LIN {X 0,Y 530.989,Z 469.465,A -85,B 0,C 180,E1 -4213.071,E2 -4213.071} C_VEL
LIN {X 0,Y 531.043,Z 469.464,A -85,B 0,C 180,E1 -4215.436,E2 -4215.436} C_VEL
LIN {X 0,Y 531.04,Z 469.456,A -85,B 0,C 180,E1 -4218.55,E2 -4218.55} C_VEL
LIN {X 0,Y 531.062,Z 469.46,A -85,B 0,C 180,E1 -4221.629,E2 -4221.629} C_VEL
LIN {X 0,Y 531.124,Z 469.446,A -85,B 0,C 180,E1 -4224.685,E2 -4224.685} C_VEL
LIN {X 0,Y 531.144,Z 469.448,A -85,B 0,C 180,E1 -4227.725,E2 -4227.725} C_VEL
LIN {X 0,Y 531.154,Z 469.442,A -85,B 0,C 180,E1 -4230.758,E2 -4230.758} C_VEL
LIN {X 0,Y 531.108,Z 469.451,A -85,B 0,C 180,E1 -4233.034,E2 -4233.034} C_VEL
LIN {X 0,Y 531.078,Z 469.452,A -85,B 0,C 180,E1 -4236.077,E2 -4236.077} C_VEL
LIN {X 0,Y 531.058,Z 469.454,A -85,B 0,C 180,E1 -4238.37,E2 -4238.37} C_VEL
LIN {X 0,Y 531.054,Z 469.459,A -85,B 0,C 180,E1 -4241.672,E2 -4241.672} C_VEL
LIN {X 0,Y 531.033,Z 469.46,A -85,B 0,C 180,E1 -4244.956,E2 -4244.956} C_VEL
LIN {X 0,Y 531.019,Z 469.463,A -85,B 0,C 180,E1 -4247.722,E2 -4247.722} C_VEL
LIN {X 0,Y 531.002,Z 469.464,A -85,B 0,C 180,E1 -4250.938,E2 -4250.938} C_VEL
LIN {X 0,Y 530.982,Z 469.463,A -85,B 0,C 180,E1 -4254.224,E2 -4254.224} C_VEL
LIN {X 0,Y 531.006,Z 469.461,A -85,B 0,C 180,E1 -4256.744,E2 -4256.744} C_VEL
LIN {X 0,Y 530.984,Z 469.472,A -85,B 0,C 180,E1 -4259.323,E2 -4259.323} C_VEL
LIN {X 0,Y 530.968,Z 469.465,A -85,B 0,C 180,E1 -4262.1,E2 -4262.1} C_VEL
LIN {X 0,Y 530.972,Z 469.467,A -85,B 0,C 180,E1 -4264.851,E2 -4264.851} C_VEL
LIN {X 0,Y 530.968,Z 469.472,A -85,B 0,C 180,E1 -4267.508,E2 -4267.508} C_VEL
LIN {X 0,Y 530.986,Z 469.463,A -85,B 0,C 180,E1 -4270.433,E2 -4270.433} C_VEL
LIN {X 0,Y 530.973,Z 469.473,A -85,B 0,C 180,E1 -4273.282,E2 -4273.282} C_VEL
LIN {X 0,Y 530.985,Z 469.467,A -85,B 0,C 180,E1 -4275.622,E2 -4275.622} C_VEL
LIN {X 0,Y 530.995,Z 469.462,A -85,B 0,C 180,E1 -4278.565,E2 -4278.565} C_VEL
LIN {X 0,Y 530.961,Z 469.471,A -85,B 0,C 180,E1 -4281.53,E2 -4281.53} C_VEL
LIN {X 0,Y 530.959,Z 469.466,A -85,B 0,C 180,E1 -4284.38,E2 -4284.38} C_VEL
LIN {X 0,Y 530.97,Z 469.472,A -85,B 0,C 180,E1 -4287.134,E2 -4287.134} C_VEL
LIN {X 0,Y 530.972,Z 469.467,A -85,B 0,C 180,E1 -4289.803,E2 -4289.803} C_VEL
LIN {X 0,Y 531.015,Z 469.461,A -85,B 0,C 180,E1 -4292.468,E2 -4292.468} C_VEL
LIN {X 0,Y 531.043,Z 469.626,A -85,B 0,C 180,E1 -4294.433,E2 -4294.433} C_VEL
LIN {X 0,Y 532.717,Z 478.043,A -85,B 0,C 180,E1 -4295.699,E2 -4295.699} C_VEL
LIN {X 0,Y 532.591,Z 490.919,A -85,B 0,C 180,E1 -4297.5,E2 -4297.5} C_VEL
LIN {X 0,Y 532.133,Z 510.715,A -85,B 0,C 180,E1 -4300.319,E2 -4300.319} C_VEL
LIN {X 0,Y 531.751,Z 532.106,A -85,B 0,C 180,E1 -4303.294,E2 -4303.294} C_VEL
LIN {X 0,Y 531.511,Z 544.809,A -85,B 0,C 180,E1 -4305.09,E2 -4305.09} C_VEL
LIN {X 0,Y 532.811,Z 554.136,A -85,B 0,C 180,E1 -4305.262,E2 -4305.262} C_VEL
LIN {X 0,Y 532.416,Z 652.888,A -85,B 0,C 180,E1 -4306.62,E2 -4306.62} C_VEL
LIN {X 0,Y 532.247,Z 665.054,A -85,B 0,C 180,E1 -4306.907,E2 -4306.907} C_VEL
LIN {X 0,Y 532.045,Z 678.792,A -85,B 0,C 180,E1 -4307.411,E2 -4307.411} C_VEL
LIN {X 0,Y 531.781,Z 689.648,A -85,B 0,C 180,E1 -4307.956,E2 -4307.956} C_VEL
LIN {X 0,Y 531.654,Z 697.634,A -85,B 0,C 180,E1 -4308.447,E2 -4308.447} C_VEL
LIN {X 0,Y 531.413,Z 706.954,A -85,B 0,C 180,E1 -4309.137,E2 -4309.137} C_VEL
LIN {X 0,Y 531.231,Z 713.575,A -85,B 0,C 180,E1 -4309.712,E2 -4309.712} C_VEL
LIN {X 0,Y 531.071,Z 721.12,A -85,B 0,C 180,E1 -4310.478,E2 -4310.478} C_VEL
LIN {X 0,Y 530.921,Z 727.6,A -85,B 0,C 180,E1 -4311.244,E2 -4311.244} C_VEL
LIN {X 0,Y 530.76,Z 734.405,A -85,B 0,C 180,E1 -4312.2,E2 -4312.2} C_VEL
LIN {X 0,Y 530.643,Z 740.091,A -85,B 0,C 180,E1 -4313.154,E2 -4313.154} C_VEL
LIN {X 0,Y 530.609,Z 745.619,A -85,B 0,C 180,E1 -4314.299,E2 -4314.299} C_VEL
LIN {X 0,Y 530.462,Z 749.968,A -85,B 0,C 180,E1 -4315.441,E2 -4315.441} C_VEL
LIN {X 0,Y 530.516,Z 752.339,A -85,B 0,C 180,E1 -4316.202,E2 -4316.202} C_VEL
LIN {X 0,Y 530.457,Z 754.172,A -85,B 0,C 180,E1 -4316.962,E2 -4316.962} C_VEL
LIN {X 0,Y 530.361,Z 756.638,A -85,B 0,C 180,E1 -4318.481,E2 -4318.481} C_VEL
LIN {X 0,Y 530.344,Z 757.24,A -85,B 0,C 180,E1 -4319.241,E2 -4319.241} C_VEL
LIN {X 0,Y 530.344,Z 757.307,A -85,B 0,C 180,E1 -4320.759,E2 -4320.759} C_VEL
LIN {X 0,Y 530.361,Z 756.712,A -85,B 0,C 180,E1 -4321.519,E2 -4321.519} C_VEL
LIN {X 0,Y 530.457,Z 754.383,A -85,B 0,C 180,E1 -4323.038,E2 -4323.038} C_VEL
LIN {X 0,Y 530.522,Z 751.5,A -85,B 0,C 180,E1 -4324.178,E2 -4324.178} C_VEL
LIN {X 0,Y 530.523,Z 747.581,A -85,B 0,C 180,E1 -4325.321,E2 -4325.321} C_VEL
LIN {X 0,Y 530.552,Z 743.338,A -85,B 0,C 180,E1 -4326.305,E2 -4326.305} C_VEL
LIN {X 0,Y 530.678,Z 737.337,A -85,B 0,C 180,E1 -4327.419,E2 -4327.419} C_VEL
LIN {X 0,Y 530.843,Z 731.101,A -85,B 0,C 180,E1 -4328.374,E2 -4328.374} C_VEL
LIN {X 0,Y 530.978,Z 723.591,A -85,B 0,C 180,E1 -4329.331,E2 -4329.331} C_VEL
LIN {X 0,Y 531.199,Z 716.488,A -85,B 0,C 180,E1 -4330.096,E2 -4330.096} C_VEL
LIN {X 0,Y 531.382,Z 708.045,A -85,B 0,C 180,E1 -4330.863,E2 -4330.863} C_VEL
LIN {X 0,Y 531.562,Z 700.597,A -85,B 0,C 180,E1 -4331.439,E2 -4331.439} C_VEL
LIN {X 0,Y 531.786,Z 691.155,A -85,B 0,C 180,E1 -4332.047,E2 -4332.047} C_VEL
LIN {X 0,Y 531.939,Z 680.692,A -85,B 0,C 180,E1 -4332.592,E2 -4332.592} C_VEL
LIN {X 0,Y 532.174,Z 669.962,A -85,B 0,C 180,E1 -4333.022,E2 -4333.022} C_VEL
LIN {X 0,Y 532.375,Z 656.359,A -85,B 0,C 180,E1 -4333.406,E2 -4333.406} C_VEL
LIN {X 0,Y 532.522,Z 634.145,A -85,B 0,C 180,E1 -4333.742,E2 -4333.742} C_VEL
LIN {X 0,Y 532.733,Z 552.911,A -85,B 0,C 180,E1 -4334.844,E2 -4334.844} C_VEL
LIN {X 0,Y 531.512,Z 544.794,A -85,B 0,C 180,E1 -4335.007,E2 -4335.007} C_VEL
LIN {X 0,Y 531.862,Z 525.613,A -85,B 0,C 180,E1 -4337.693,E2 -4337.693} C_VEL
LIN {X 0,Y 532.252,Z 507.489,A -85,B 0,C 180,E1 -4340.244,E2 -4340.244} C_VEL
LIN {X 0,Y 532.568,Z 484.627,A -85,B 0,C 180,E1 -4343.322,E2 -4343.322} C_VEL
LIN {X 0,Y 532.427,Z 476.639,A -85,B 0,C 180,E1 -4344.384,E2 -4344.384} C_VEL
LIN {X 0,Y 531.039,Z 469.463,A -85,B 0,C 180,E1 -4345.423,E2 -4345.423} C_VEL
LIN {X 0,Y 531,Z 469.469,A -85,B 0,C 180,E1 -4348.455,E2 -4348.455} C_VEL
LIN {X 0,Y 530.96,Z 469.474,A -85,B 0,C 180,E1 -4351.079,E2 -4351.079} C_VEL
LIN {X 0,Y 530.99,Z 469.465,A -85,B 0,C 180,E1 -4353.773,E2 -4353.773} C_VEL
LIN {X 0,Y 530.958,Z 469.475,A -85,B 0,C 180,E1 -4356.558,E2 -4356.558} C_VEL
LIN {X 0,Y 530.991,Z 469.464,A -85,B 0,C 180,E1 -4359.443,E2 -4359.443} C_VEL
LIN {X 0,Y 530.98,Z 469.471,A -85,B 0,C 180,E1 -4362.457,E2 -4362.457} C_VEL
LIN {X 0,Y 530.991,Z 469.463,A -85,B 0,C 180,E1 -4365.621,E2 -4365.621} C_VEL
LIN {X 0,Y 531,Z 469.469,A -85,B 0,C 180,E1 -4368.565,E2 -4368.565} C_VEL
LIN {X 0,Y 530.96,Z 469.467,A -85,B 0,C 180,E1 -4371.529,E2 -4371.529} C_VEL
LIN {X 0,Y 530.982,Z 469.471,A -85,B 0,C 180,E1 -4374.382,E2 -4374.382} C_VEL
LIN {X 0,Y 530.975,Z 469.466,A -85,B 0,C 180,E1 -4377.134,E2 -4377.134} C_VEL
LIN {X 0,Y 530.989,Z 469.467,A -85,B 0,C 180,E1 -4379.804,E2 -4379.804} C_VEL
LIN {X 0,Y 531.017,Z 469.468,A -85,B 0,C 180,E1 -4382.467,E2 -4382.467} C_VEL
LIN {X 0,Y 531.078,Z 469.651,A -85,B 0,C 180,E1 -4384.92,E2 -4384.92} C_VEL
LIN {X 0,Y 533.286,Z 479.428,A -85,B 0,C 180,E1 -4386.3,E2 -4386.3} C_VEL
LIN {X 0,Y 532.933,Z 495.381,A -85,B 0,C 180,E1 -4388.331,E2 -4388.331} C_VEL
LIN {X 0,Y 532.3,Z 520.903,A -85,B 0,C 180,E1 -4391.526,E2 -4391.526} C_VEL
LIN {X 0,Y 532.17,Z 524.017,A -85,B 0,C 180,E1 -4391.91,E2 -4391.91} C_VEL
LIN {X 0,Y 533.88,Z 534.449,A -85,B 0,C 180,E1 -4392.114,E2 -4392.114} C_VEL
LIN {X 0,Y 533.255,Z 662.06,A -85,B 0,C 180,E1 -4393.859,E2 -4393.859} C_VEL
LIN {X 0,Y 533.024,Z 676.356,A -85,B 0,C 180,E1 -4394.202,E2 -4394.202} C_VEL
LIN {X 0,Y 532.797,Z 690.478,A -85,B 0,C 180,E1 -4394.703,E2 -4394.703} C_VEL
LIN {X 0,Y 532.549,Z 702.8,A -85,B 0,C 180,E1 -4395.283,E2 -4395.283} C_VEL
LIN {X 0,Y 532.13,Z 715.67,A -85,B 0,C 180,E1 -4396.052,E2 -4396.052} C_VEL
LIN {X 0,Y 531.813,Z 727.305,A -85,B 0,C 180,E1 -4396.92,E2 -4396.92} C_VEL
LIN {X 0,Y 531.463,Z 738.313,A -85,B 0,C 180,E1 -4397.917,E2 -4397.917} C_VEL
LIN {X 0,Y 531.235,Z 747.706,A -85,B 0,C 180,E1 -4398.94,E2 -4398.94} C_VEL
LIN {X 0,Y 530.935,Z 756.556,A -85,B 0,C 180,E1 -4400.091,E2 -4400.091} C_VEL
LIN {X 0,Y 530.775,Z 765.034,A -85,B 0,C 180,E1 -4401.433,E2 -4401.433} C_VEL
LIN {X 0,Y 530.586,Z 771.863,A -85,B 0,C 180,E1 -4402.771,E2 -4402.771} C_VEL
LIN {X 0,Y 530.584,Z 777.961,A -85,B 0,C 180,E1 -4404.299,E2 -4404.299} C_VEL
LIN {X 0,Y 530.449,Z 781.444,A -85,B 0,C 180,E1 -4405.44,E2 -4405.44} C_VEL
LIN {X 0,Y 530.452,Z 784.832,A -85,B 0,C 180,E1 -4406.962,E2 -4406.962} C_VEL
LIN {X 0,Y 530.356,Z 786.835,A -85,B 0,C 180,E1 -4408.481,E2 -4408.481} C_VEL
LIN {X 0,Y 530.341,Z 787.5,A -85,B 0,C 180,E1 -4410,E2 -4410} C_VEL
LIN {X 0,Y 530.356,Z 786.836,A -85,B 0,C 180,E1 -4411.519,E2 -4411.519} C_VEL
LIN {X 0,Y 530.452,Z 784.836,A -85,B 0,C 180,E1 -4413.038,E2 -4413.038} C_VEL
LIN {X 0,Y 530.449,Z 781.446,A -85,B 0,C 180,E1 -4414.56,E2 -4414.56} C_VEL
LIN {X 0,Y 530.56,Z 776.567,A -85,B 0,C 180,E1 -4416.083,E2 -4416.083} C_VEL
LIN {X 0,Y 530.641,Z 770.053,A -85,B 0,C 180,E1 -4417.611,E2 -4417.611} C_VEL
LIN {X 0,Y 530.818,Z 762.803,A -85,B 0,C 180,E1 -4418.95,E2 -4418.95} C_VEL
LIN {X 0,Y 531.018,Z 753.821,A -85,B 0,C 180,E1 -4420.293,E2 -4420.293} C_VEL
LIN {X 0,Y 531.311,Z 744.391,A -85,B 0,C 180,E1 -4421.444,E2 -4421.444} C_VEL
LIN {X 0,Y 531.585,Z 733.95,A -85,B 0,C 180,E1 -4422.503,E2 -4422.503} C_VEL
LIN {X 0,Y 531.956,Z 722.424,A -85,B 0,C 180,E1 -4423.465,E2 -4423.465} C_VEL
LIN {X 0,Y 532.29,Z 709.619,A -85,B 0,C 180,E1 -4424.333,E2 -4424.333} C_VEL
LIN {X 0,Y 532.625,Z 696.975,A -85,B 0,C 180,E1 -4425.008,E2 -4425.008} C_VEL
LIN {X 0,Y 532.891,Z 683.069,A -85,B 0,C 180,E1 -4425.579,E2 -4425.579} C_VEL
LIN {X 0,Y 533.151,Z 668.504,A -85,B 0,C 180,E1 -4426.002,E2 -4426.002} C_VEL
LIN {X 0,Y 533.291,Z 653.936,A -85,B 0,C 180,E1 -4426.263,E2 -4426.263} C_VEL
LIN {X 0,Y 533.831,Z 534.167,A -85,B 0,C 180,E1 -4427.883,E2 -4427.883} C_VEL
LIN {X 0,Y 532.175,Z 524.02,A -85,B 0,C 180,E1 -4428.083,E2 -4428.083} C_VEL
LIN {X 0,Y 532.831,Z 498.464,A -85,B 0,C 180,E1 -4431.268,E2 -4431.268} C_VEL
LIN {X 0,Y 533.425,Z 481.072,A -85,B 0,C 180,E1 -4433.488,E2 -4433.488} C_VEL
LIN {X 0,Y 532.289,Z 474.884,A -85,B 0,C 180,E1 -4434.352,E2 -4434.352} C_VEL
LIN {X 0,Y 531.038,Z 469.465,A -85,B 0,C 180,E1 -4435.161,E2 -4435.161} C_VEL
LIN {X 0,Y 531.018,Z 469.468,A -85,B 0,C 180,E1 -4437.596,E2 -4437.596} C_VEL
LIN {X 0,Y 530.978,Z 469.468,A -85,B 0,C 180,E1 -4440.645,E2 -4440.645} C_VEL
LIN {X 0,Y 530.989,Z 469.47,A -85,B 0,C 180,E1 -4443.773,E2 -4443.773} C_VEL
LIN {X 0,Y 530.957,Z 469.469,A -85,B 0,C 180,E1 -4446.559,E2 -4446.559} C_VEL
LIN {X 0,Y 530.989,Z 469.471,A -85,B 0,C 180,E1 -4449.444,E2 -4449.444} C_VEL
LIN {X 0,Y 530.984,Z 469.465,A -85,B 0,C 180,E1 -4452.457,E2 -4452.457} C_VEL
LIN {X 0,Y 530.985,Z 469.467,A -85,B 0,C 180,E1 -4455.622,E2 -4455.622} C_VEL
LIN {X 0,Y 530.999,Z 469.466,A -85,B 0,C 180,E1 -4458.565,E2 -4458.565} C_VEL
LIN {X 0,Y 530.963,Z 469.47,A -85,B 0,C 180,E1 -4461.53,E2 -4461.53} C_VEL
LIN {X 0,Y 530.962,Z 469.471,A -85,B 0,C 180,E1 -4464.38,E2 -4464.38} C_VEL
LIN {X 0,Y 530.975,Z 469.471,A -85,B 0,C 180,E1 -4467.134,E2 -4467.134} C_VEL
LIN {X 0,Y 530.974,Z 469.468,A -85,B 0,C 180,E1 -4469.803,E2 -4469.803} C_VEL
LIN {X 0,Y 531.019,Z 469.471,A -85,B 0,C 180,E1 -4472.467,E2 -4472.467} C_VEL
LIN {X 0,Y 531.028,Z 469.511,A -85,B 0,C 180,E1 -4475.413,E2 -4475.413} C_VEL
LIN {X 0,Y 532.922,Z 478.715,A -85,B 0,C 180,E1 -4476.9,E2 -4476.9} C_VEL
LIN {X 0,Y 532.484,Z 495.757,A -85,B 0,C 180,E1 -4479.422,E2 -4479.422} C_VEL
LIN {X 0,Y 531.978,Z 516.977,A -85,B 0,C 180,E1 -4482.509,E2 -4482.509} C_VEL
LIN {X 0,Y 531.53,Z 538.766,A -85,B 0,C 180,E1 -4485.646,E2 -4485.646} C_VEL
LIN {X 0,Y 531.459,Z 541.741,A -85,B 0,C 180,E1 -4486.071,E2 -4486.071} C_VEL
LIN {X 0,Y 532.832,Z 550.807,A -85,B 0,C 180,E1 -4486.241,E2 -4486.241} C_VEL
LIN {X 0,Y 532.381,Z 651.089,A -85,B 0,C 180,E1 -4487.632,E2 -4487.632} C_VEL
LIN {X 0,Y 532.255,Z 663.912,A -85,B 0,C 180,E1 -4487.964,E2 -4487.964} C_VEL
LIN {X 0,Y 532.036,Z 675.604,A -85,B 0,C 180,E1 -4488.399,E2 -4488.399} C_VEL
LIN {X 0,Y 531.878,Z 686.69,A -85,B 0,C 180,E1 -4488.954,E2 -4488.954} C_VEL
LIN {X 0,Y 531.586,Z 697.237,A -85,B 0,C 180,E1 -4489.622,E2 -4489.622} C_VEL
LIN {X 0,Y 531.354,Z 707.051,A -85,B 0,C 180,E1 -4490.387,E2 -4490.387} C_VEL
LIN {X 0,Y 531.088,Z 717.832,A -85,B 0,C 180,E1 -4491.438,E2 -4491.438} C_VEL
LIN {X 0,Y 530.861,Z 725.753,A -85,B 0,C 180,E1 -4492.392,E2 -4492.392} C_VEL
LIN {X 0,Y 530.739,Z 733.573,A -85,B 0,C 180,E1 -4493.537,E2 -4493.537} C_VEL
LIN {X 0,Y 530.55,Z 739.838,A -85,B 0,C 180,E1 -4494.68,E2 -4494.68} C_VEL
LIN {X 0,Y 530.558,Z 744.79,A -85,B 0,C 180,E1 -4495.822,E2 -4495.822} C_VEL
LIN {X 0,Y 530.509,Z 748.671,A -85,B 0,C 180,E1 -4496.962,E2 -4496.962} C_VEL
LIN {X 0,Y 530.432,Z 750.661,A -85,B 0,C 180,E1 -4497.722,E2 -4497.722} C_VEL
LIN {X 0,Y 530.366,Z 752.216,A -85,B 0,C 180,E1 -4498.481,E2 -4498.481} C_VEL
LIN {X 0,Y 530.345,Z 753.356,A -85,B 0,C 180,E1 -4499.241,E2 -4499.241} C_VEL
LIN {X 0,Y 530.344,Z 754.095,A -85,B 0,C 180,E1 -4500,E2 -4500} C_VEL
LIN {X 0,Y 530.361,Z 754.383,A -85,B 0,C 180,E1 -4501.519,E2 -4501.519} C_VEL
LIN {X 0,Y 530.409,Z 753.938,A -85,B 0,C 180,E1 -4502.278,E2 -4502.278} C_VEL
LIN {X 0,Y 530.452,Z 753.091,A -85,B 0,C 180,E1 -4503.038,E2 -4503.038} C_VEL
LIN {X 0,Y 530.488,Z 751.84,A -85,B 0,C 180,E1 -4503.798,E2 -4503.798} C_VEL
LIN {X 0,Y 530.438,Z 749.208,A -85,B 0,C 180,E1 -4504.94,E2 -4504.94} C_VEL
LIN {X 0,Y 530.513,Z 745.486,A -85,B 0,C 180,E1 -4506.084,E2 -4506.084} C_VEL
LIN {X 0,Y 530.577,Z 740.727,A -85,B 0,C 180,E1 -4507.229,E2 -4507.229} C_VEL
LIN {X 0,Y 530.706,Z 734.613,A -85,B 0,C 180,E1 -4508.376,E2 -4508.376} C_VEL
LIN {X 0,Y 530.837,Z 727.039,A -85,B 0,C 180,E1 -4509.526,E2 -4509.526} C_VEL
LIN {X 0,Y 531.051,Z 719.353,A -85,B 0,C 180,E1 -4510.484,E2 -4510.484} C_VEL
LIN {X 0,Y 531.254,Z 709.888,A -85,B 0,C 180,E1 -4511.446,E2 -4511.446} C_VEL
LIN {X 0,Y 531.528,Z 699.399,A -85,B 0,C 180,E1 -4512.31,E2 -4512.31} C_VEL
LIN {X 0,Y 531.782,Z 689.383,A -85,B 0,C 180,E1 -4512.984,E2 -4512.984} C_VEL
LIN {X 0,Y 531.979,Z 677.385,A -85,B 0,C 180,E1 -4513.611,E2 -4513.611} C_VEL
LIN {X 0,Y 532.2,Z 664.294,A -85,B 0,C 180,E1 -4514.116,E2 -4514.116} C_VEL
LIN {X 0,Y 532.38,Z 652.592,A -85,B 0,C 180,E1 -4514.428,E2 -4514.428} C_VEL
LIN {X 0,Y 532.561,Z 626.378,A -85,B 0,C 180,E1 -4514.814,E2 -4514.814} C_VEL
LIN {X 0,Y 532.691,Z 549.68,A -85,B 0,C 180,E1 -4515.866,E2 -4515.866} C_VEL
LIN {X 0,Y 531.451,Z 541.613,A -85,B 0,C 180,E1 -4516.035,E2 -4516.035} C_VEL
LIN {X 0,Y 531.894,Z 521.744,A -85,B 0,C 180,E1 -4518.888,E2 -4518.888} C_VEL
LIN {X 0,Y 532.357,Z 501.091,A -85,B 0,C 180,E1 -4521.893,E2 -4521.893} C_VEL
LIN {X 0,Y 532.912,Z 481.342,A -85,B 0,C 180,E1 -4524.809,E2 -4524.809} C_VEL
LIN {X 0,Y 532.756,Z 477.549,A -85,B 0,C 180,E1 -4525.387,E2 -4525.387} C_VEL
LIN {X 0,Y 532.142,Z 474.583,A -85,B 0,C 180,E1 -4525.866,E2 -4525.866} C_VEL
LIN {X 0,Y 531.021,Z 472.733,A -85,B 0,C 180,E1 -4526.232,E2 -4526.232} C_VEL
LIN {X 0,Y 529.133,Z 471.526,A -85,B 0,C 180,E1 -4526.602,E2 -4526.602} C_VEL
LIN {X 0,Y 526.354,Z 470.672,A -85,B 0,C 180,E1 -4527.107,E2 -4527.107} C_VEL
LIN {X 0,Y 524.307,Z 470.372,A -85,B 0,C 180,E1 -4527.657,E2 -4527.657} C_VEL
LIN {X 0,Y 523.972,Z 470.345,A -85,B 0,C 180,E1 -4527.95,E2 -4527.95} C_VEL
LIN {X 0,Y 523.948,Z 470.343,A -85,B 0,C 180,E1 -4530.855,E2 -4530.855} C_VEL
LIN {X 0,Y 523.964,Z 470.346,A -85,B 0,C 180,E1 -4533.735,E2 -4533.735} C_VEL
LIN {X 0,Y 523.911,Z 470.345,A -85,B 0,C 180,E1 -4536.402,E2 -4536.402} C_VEL
LIN {X 0,Y 523.924,Z 470.344,A -85,B 0,C 180,E1 -4539.084,E2 -4539.084} C_VEL
LIN {X 0,Y 523.954,Z 470.341,A -85,B 0,C 180,E1 -4542.119,E2 -4542.119} C_VEL
LIN {X 0,Y 523.949,Z 470.344,A -85,B 0,C 180,E1 -4545.31,E2 -4545.31} C_VEL
LIN {X 0,Y 523.961,Z 470.338,A -85,B 0,C 180,E1 -4548.689,E2 -4548.689} C_VEL
LIN {X 0,Y 523.92,Z 470.345,A -85,B 0,C 180,E1 -4551.08,E2 -4551.08} C_VEL
LIN {X 0,Y 523.903,Z 470.35,A -85,B 0,C 180,E1 -4553.825,E2 -4553.825} C_VEL
LIN {X 0,Y 523.943,Z 470.34,A -85,B 0,C 180,E1 -4556.635,E2 -4556.635} C_VEL
LIN {X 0,Y 523.958,Z 470.345,A -85,B 0,C 180,E1 -4559.356,E2 -4559.356} C_VEL
LIN {X 0,Y 523.979,Z 470.336,A -85,B 0,C 180,E1 -4562.281,E2 -4562.281} C_VEL
LIN {X 0,Y 523.955,Z 470.338,A -85,B 0,C 180,E1 -4564.581,E2 -4564.581} C_VEL
LIN {X 0,Y 523.913,Z 470.347,A -85,B 0,C 180,E1 -4567.106,E2 -4567.106} C_VEL
LIN {X 0,Y 523.981,Z 470.339,A -85,B 0,C 180,E1 -4569.866,E2 -4569.866} C_VEL
LIN {X 0,Y 523.97,Z 470.338,A -85,B 0,C 180,E1 -4572.837,E2 -4572.837} C_VEL
LIN {X 0,Y 524.007,Z 470.337,A -85,B 0,C 180,E1 -4575.236,E2 -4575.236} C_VEL
LIN {X 0,Y 524.015,Z 470.331,A -85,B 0,C 180,E1 -4578.394,E2 -4578.394} C_VEL
LIN {X 0,Y 524.01,Z 470.341,A -85,B 0,C 180,E1 -4581.516,E2 -4581.516} C_VEL
LIN {X 0,Y 524.085,Z 470.322,A -85,B 0,C 180,E1 -4584.614,E2 -4584.614} C_VEL
LIN {X 0,Y 524.116,Z 470.324,A -85,B 0,C 180,E1 -4587.694,E2 -4587.694} C_VEL
LIN {X 0,Y 524.125,Z 470.318,A -85,B 0,C 180,E1 -4590.768,E2 -4590.768} C_VEL
LIN {X 0,Y 524.075,Z 470.327,A -85,B 0,C 180,E1 -4593.075,E2 -4593.075} C_VEL
LIN {X 0,Y 524.04,Z 470.328,A -85,B 0,C 180,E1 -4596.159,E2 -4596.159} C_VEL
LIN {X 0,Y 524.006,Z 470.332,A -85,B 0,C 180,E1 -4598.484,E2 -4598.484} C_VEL
LIN {X 0,Y 524.005,Z 470.337,A -85,B 0,C 180,E1 -4601.74,E2 -4601.74} C_VEL
LIN {X 0,Y 523.995,Z 470.338,A -85,B 0,C 180,E1 -4605.052,E2 -4605.052} C_VEL
LIN {X 0,Y 523.966,Z 470.339,A -85,B 0,C 180,E1 -4607.969,E2 -4607.969} C_VEL
LIN {X 0,Y 523.974,Z 470.336,A -85,B 0,C 180,E1 -4610.41,E2 -4610.41} C_VEL
LIN {X 0,Y 523.919,Z 470.345,A -85,B 0,C 180,E1 -4612.893,E2 -4612.893} C_VEL
LIN {X 0,Y 523.956,Z 470.347,A -85,B 0,C 180,E1 -4615.419,E2 -4615.419} C_VEL
LIN {X 0,Y 523.971,Z 470.338,A -85,B 0,C 180,E1 -4617.999,E2 -4617.999} C_VEL
LIN {X 0,Y 523.947,Z 470.342,A -85,B 0,C 180,E1 -4620.855,E2 -4620.855} C_VEL
LIN {X 0,Y 523.961,Z 470.341,A -85,B 0,C 180,E1 -4623.734,E2 -4623.734} C_VEL
LIN {X 0,Y 523.905,Z 470.345,A -85,B 0,C 180,E1 -4626.401,E2 -4626.401} C_VEL
LIN {X 0,Y 523.925,Z 470.348,A -85,B 0,C 180,E1 -4629.085,E2 -4629.085} C_VEL
LIN {X 0,Y 523.96,Z 470.338,A -85,B 0,C 180,E1 -4632.118,E2 -4632.118} C_VEL
LIN {X 0,Y 523.955,Z 470.348,A -85,B 0,C 180,E1 -4635.309,E2 -4635.309} C_VEL
LIN {X 0,Y 523.958,Z 470.34,A -85,B 0,C 180,E1 -4638.69,E2 -4638.69} C_VEL
LIN {X 0,Y 523.921,Z 470.349,A -85,B 0,C 180,E1 -4641.08,E2 -4641.08} C_VEL
LIN {X 0,Y 523.903,Z 470.347,A -85,B 0,C 180,E1 -4643.825,E2 -4643.825} C_VEL
LIN {X 0,Y 523.944,Z 470.341,A -85,B 0,C 180,E1 -4646.636,E2 -4646.636} C_VEL
LIN {X 0,Y 523.958,Z 470.346,A -85,B 0,C 180,E1 -4649.356,E2 -4649.356} C_VEL
LIN {X 0,Y 523.98,Z 470.337,A -85,B 0,C 180,E1 -4652.282,E2 -4652.282} C_VEL
LIN {X 0,Y 523.988,Z 470.355,A -85,B 0,C 180,E1 -4654.226,E2 -4654.226} C_VEL
LIN {X 0,Y 525.879,Z 480.356,A -85,B 0,C 180,E1 -4655.735,E2 -4655.735} C_VEL
LIN {X 0,Y 525.511,Z 499.272,A -85,B 0,C 180,E1 -4658.422,E2 -4658.422} C_VEL
LIN {X 0,Y 525.02,Z 522.036,A -85,B 0,C 180,E1 -4661.654,E2 -4661.654} C_VEL
LIN {X 0,Y 524.589,Z 541.882,A -85,B 0,C 180,E1 -4664.458,E2 -4664.458} C_VEL
LIN {X 0,Y 524.523,Z 544.936,A -85,B 0,C 180,E1 -4664.895,E2 -4664.895} C_VEL
LIN {X 0,Y 525.926,Z 555.452,A -85,B 0,C 180,E1 -4665.089,E2 -4665.089} C_VEL
LIN {X 0,Y 525.49,Z 653.567,A -85,B 0,C 180,E1 -4666.464,E2 -4666.464} C_VEL
LIN {X 0,Y 525.313,Z 666.27,A -85,B 0,C 180,E1 -4666.78,E2 -4666.78} C_VEL
LIN {X 0,Y 525.085,Z 678.581,A -85,B 0,C 180,E1 -4667.241,E2 -4667.241} C_VEL
LIN {X 0,Y 524.82,Z 690.335,A -85,B 0,C 180,E1 -4667.841,E2 -4667.841} C_VEL
LIN {X 0,Y 524.604,Z 700.641,A -85,B 0,C 180,E1 -4668.505,E2 -4668.505} C_VEL
LIN {X 0,Y 524.295,Z 711.545,A -85,B 0,C 180,E1 -4669.379,E2 -4669.379} C_VEL
LIN {X 0,Y 524.067,Z 721.162,A -85,B 0,C 180,E1 -4670.35,E2 -4670.35} C_VEL
LIN {X 0,Y 523.855,Z 729.065,A -85,B 0,C 180,E1 -4671.319,E2 -4671.319} C_VEL
LIN {X 0,Y 523.667,Z 735.634,A -85,B 0,C 180,E1 -4672.287,E2 -4672.287} C_VEL
LIN {X 0,Y 523.579,Z 740.124,A -85,B 0,C 180,E1 -4673.061,E2 -4673.061} C_VEL
LIN {X 0,Y 523.541,Z 745.632,A -85,B 0,C 180,E1 -4674.222,E2 -4674.222} C_VEL
LIN {X 0,Y 523.366,Z 749.964,A -85,B 0,C 180,E1 -4675.379,E2 -4675.379} C_VEL
LIN {X 0,Y 523.444,Z 752.334,A -85,B 0,C 180,E1 -4676.151,E2 -4676.151} C_VEL
LIN {X 0,Y 523.368,Z 754.167,A -85,B 0,C 180,E1 -4676.921,E2 -4676.921} C_VEL
LIN {X 0,Y 523.275,Z 756.632,A -85,B 0,C 180,E1 -4678.461,E2 -4678.461} C_VEL
LIN {X 0,Y 523.25,Z 757.233,A -85,B 0,C 180,E1 -4679.23,E2 -4679.23} C_VEL
LIN {X 0,Y 523.25,Z 757.3,A -85,B 0,C 180,E1 -4680.77,E2 -4680.77} C_VEL
LIN {X 0,Y 523.274,Z 756.705,A -85,B 0,C 180,E1 -4681.539,E2 -4681.539} C_VEL
LIN {X 0,Y 523.368,Z 754.377,A -85,B 0,C 180,E1 -4683.079,E2 -4683.079} C_VEL
LIN {X 0,Y 523.441,Z 751.493,A -85,B 0,C 180,E1 -4684.235,E2 -4684.235} C_VEL
LIN {X 0,Y 523.463,Z 747.582,A -85,B 0,C 180,E1 -4685.393,E2 -4685.393} C_VEL
LIN {X 0,Y 523.517,Z 742.427,A -85,B 0,C 180,E1 -4686.574,E2 -4686.574} C_VEL
LIN {X 0,Y 523.625,Z 737.37,A -85,B 0,C 180,E1 -4687.519,E2 -4687.519} C_VEL
LIN {X 0,Y 523.812,Z 731.141,A -85,B 0,C 180,E1 -4688.487,E2 -4688.487} C_VEL
LIN {X 0,Y 523.958,Z 723.629,A -85,B 0,C 180,E1 -4689.457,E2 -4689.457} C_VEL
LIN {X 0,Y 524.209,Z 714.52,A -85,B 0,C 180,E1 -4690.428,E2 -4690.428} C_VEL
LIN {X 0,Y 524.503,Z 704.461,A -85,B 0,C 180,E1 -4691.301,E2 -4691.301} C_VEL
LIN {X 0,Y 524.782,Z 693.254,A -85,B 0,C 180,E1 -4692.077,E2 -4692.077} C_VEL
LIN {X 0,Y 524.97,Z 681.469,A -85,B 0,C 180,E1 -4692.712,E2 -4692.712} C_VEL
LIN {X 0,Y 525.261,Z 669.509,A -85,B 0,C 180,E1 -4693.197,E2 -4693.197} C_VEL
LIN {X 0,Y 525.427,Z 656.54,A -85,B 0,C 180,E1 -4693.562,E2 -4693.562} C_VEL
LIN {X 0,Y 525.609,Z 634.354,A -85,B 0,C 180,E1 -4693.902,E2 -4693.902} C_VEL
LIN {X 0,Y 525.901,Z 553.897,A -85,B 0,C 180,E1 -4695.026,E2 -4695.026} C_VEL
LIN {X 0,Y 524.538,Z 544.88,A -85,B 0,C 180,E1 -4695.211,E2 -4695.211} C_VEL
LIN {X 0,Y 524.848,Z 528.402,A -85,B 0,C 180,E1 -4697.535,E2 -4697.535} C_VEL
LIN {X 0,Y 525.207,Z 512.818,A -85,B 0,C 180,E1 -4699.748,E2 -4699.748} C_VEL
LIN {X 0,Y 525.534,Z 490.071,A -85,B 0,C 180,E1 -4702.819,E2 -4702.819} C_VEL
LIN {X 0,Y 525.635,Z 479.289,A -85,B 0,C 180,E1 -4704.277,E2 -4704.277} C_VEL
LIN {X 0,Y 524.02,Z 470.337,A -85,B 0,C 180,E1 -4705.549,E2 -4705.549} C_VEL
LIN {X 0,Y 523.971,Z 470.341,A -85,B 0,C 180,E1 -4707.999,E2 -4707.999} C_VEL
LIN {X 0,Y 523.947,Z 470.349,A -85,B 0,C 180,E1 -4710.855,E2 -4710.855} C_VEL
LIN {X 0,Y 523.962,Z 470.341,A -85,B 0,C 180,E1 -4713.734,E2 -4713.734} C_VEL
LIN {X 0,Y 523.906,Z 470.352,A -85,B 0,C 180,E1 -4716.401,E2 -4716.401} C_VEL
LIN {X 0,Y 523.925,Z 470.347,A -85,B 0,C 180,E1 -4719.084,E2 -4719.084} C_VEL
LIN {X 0,Y 523.953,Z 470.343,A -85,B 0,C 180,E1 -4722.119,E2 -4722.119} C_VEL
LIN {X 0,Y 523.958,Z 470.339,A -85,B 0,C 180,E1 -4725.309,E2 -4725.309} C_VEL
LIN {X 0,Y 523.962,Z 470.344,A -85,B 0,C 180,E1 -4728.689,E2 -4728.689} C_VEL
LIN {X 0,Y 523.918,Z 470.347,A -85,B 0,C 180,E1 -4731.898,E2 -4731.898} C_VEL
LIN {X 0,Y 523.938,Z 470.345,A -85,B 0,C 180,E1 -4734.909,E2 -4734.909} C_VEL
LIN {X 0,Y 523.946,Z 470.342,A -85,B 0,C 180,E1 -4737.678,E2 -4737.678} C_VEL
LIN {X 0,Y 523.966,Z 470.344,A -85,B 0,C 180,E1 -4740.675,E2 -4740.675} C_VEL
LIN {X 0,Y 523.977,Z 470.343,A -85,B 0,C 180,E1 -4743.729,E2 -4743.729} C_VEL
LIN {X 0,Y 524.017,Z 470.495,A -85,B 0,C 180,E1 -4744.672,E2 -4744.672} C_VEL
LIN {X 0,Y 526.423,Z 481.01,A -85,B 0,C 180,E1 -4746.181,E2 -4746.181} C_VEL
LIN {X 0,Y 526.169,Z 493.773,A -85,B 0,C 180,E1 -4747.831,E2 -4747.831} C_VEL
LIN {X 0,Y 525.446,Z 517.7,A -85,B 0,C 180,E1 -4750.871,E2 -4750.871} C_VEL
LIN {X 0,Y 525.262,Z 524.116,A -85,B 0,C 180,E1 -4751.683,E2 -4751.683} C_VEL
LIN {X 0,Y 527.084,Z 535.152,A -85,B 0,C 180,E1 -4751.911,E2 -4751.911} C_VEL
LIN {X 0,Y 526.37,Z 660.081,A -85,B 0,C 180,E1 -4753.642,E2 -4753.642} C_VEL
LIN {X 0,Y 526.128,Z 674.91,A -85,B 0,C 180,E1 -4753.98,E2 -4753.98} C_VEL
LIN {X 0,Y 525.947,Z 688.249,A -85,B 0,C 180,E1 -4754.44,E2 -4754.44} C_VEL
LIN {X 0,Y 525.642,Z 700.246,A -85,B 0,C 180,E1 -4754.986,E2 -4754.986} C_VEL
LIN {X 0,Y 525.237,Z 713.689,A -85,B 0,C 180,E1 -4755.767,E2 -4755.767} C_VEL
LIN {X 0,Y 524.853,Z 725.761,A -85,B 0,C 180,E1 -4756.645,E2 -4756.645} C_VEL
LIN {X 0,Y 524.543,Z 736.766,A -85,B 0,C 180,E1 -4757.621,E2 -4757.621} C_VEL
LIN {X 0,Y 524.227,Z 747.616,A -85,B 0,C 180,E1 -4758.791,E2 -4758.791} C_VEL
LIN {X 0,Y 523.903,Z 756.55,A -85,B 0,C 180,E1 -4759.957,E2 -4759.957} C_VEL
LIN {X 0,Y 523.728,Z 763.918,A -85,B 0,C 180,E1 -4761.123,E2 -4761.123} C_VEL
LIN {X 0,Y 523.569,Z 770.054,A -85,B 0,C 180,E1 -4762.286,E2 -4762.286} C_VEL
LIN {X 0,Y 523.473,Z 776.569,A -85,B 0,C 180,E1 -4763.834,E2 -4763.834} C_VEL
LIN {X 0,Y 523.376,Z 780.38,A -85,B 0,C 180,E1 -4764.993,E2 -4764.993} C_VEL
LIN {X 0,Y 523.419,Z 783.316,A -85,B 0,C 180,E1 -4766.151,E2 -4766.151} C_VEL
LIN {X 0,Y 523.332,Z 786.003,A -85,B 0,C 180,E1 -4767.691,E2 -4767.691} C_VEL
LIN {X 0,Y 523.247,Z 787.334,A -85,B 0,C 180,E1 -4769.23,E2 -4769.23} C_VEL
LIN {X 0,Y 523.247,Z 787.334,A -85,B 0,C 180,E1 -4770.77,E2 -4770.77} C_VEL
LIN {X 0,Y 523.332,Z 786.005,A -85,B 0,C 180,E1 -4772.309,E2 -4772.309} C_VEL
LIN {X 0,Y 523.419,Z 783.32,A -85,B 0,C 180,E1 -4773.85,E2 -4773.85} C_VEL
LIN {X 0,Y 523.452,Z 779.201,A -85,B 0,C 180,E1 -4775.393,E2 -4775.393} C_VEL
LIN {X 0,Y 523.495,Z 773.526,A -85,B 0,C 180,E1 -4776.94,E2 -4776.94} C_VEL
LIN {X 0,Y 523.665,Z 767.126,A -85,B 0,C 180,E1 -4778.295,E2 -4778.295} C_VEL
LIN {X 0,Y 523.863,Z 759.173,A -85,B 0,C 180,E1 -4779.654,E2 -4779.654} C_VEL
LIN {X 0,Y 524.118,Z 750.792,A -85,B 0,C 180,E1 -4780.82,E2 -4780.82} C_VEL
LIN {X 0,Y 524.428,Z 740.903,A -85,B 0,C 180,E1 -4781.96,E2 -4781.96} C_VEL
LIN {X 0,Y 524.678,Z 730.377,A -85,B 0,C 180,E1 -4782.966,E2 -4782.966} C_VEL
LIN {X 0,Y 525.031,Z 719.269,A -85,B 0,C 180,E1 -4783.844,E2 -4783.844} C_VEL
LIN {X 0,Y 525.413,Z 707.21,A -85,B 0,C 180,E1 -4784.624,E2 -4784.624} C_VEL
LIN {X 0,Y 525.738,Z 693.859,A -85,B 0,C 180,E1 -4785.309,E2 -4785.309} C_VEL
LIN {X 0,Y 526.046,Z 680.005,A -85,B 0,C 180,E1 -4785.844,E2 -4785.844} C_VEL
LIN {X 0,Y 526.271,Z 666.655,A -85,B 0,C 180,E1 -4786.211,E2 -4786.211} C_VEL
LIN {X 0,Y 526.42,Z 648.922,A -85,B 0,C 180,E1 -4786.506,E2 -4786.506} C_VEL
LIN {X 0,Y 526.956,Z 534.532,A -85,B 0,C 180,E1 -4788.084,E2 -4788.084} C_VEL
LIN {X 0,Y 525.289,Z 524.092,A -85,B 0,C 180,E1 -4788.311,E2 -4788.311} C_VEL
LIN {X 0,Y 525.947,Z 500.048,A -85,B 0,C 180,E1 -4791.354,E2 -4791.354} C_VEL
LIN {X 0,Y 526.587,Z 482.677,A -85,B 0,C 180,E1 -4793.603,E2 -4793.603} C_VEL
LIN {X 0,Y 525.35,Z 476.164,A -85,B 0,C 180,E1 -4794.538,E2 -4794.538} C_VEL
LIN {X 0,Y 523.99,Z 470.343,A -85,B 0,C 180,E1 -4795.417,E2 -4795.417} C_VEL
LIN {X 0,Y 523.972,Z 470.346,A -85,B 0,C 180,E1 -4797.999,E2 -4797.999} C_VEL
LIN {X 0,Y 523.95,Z 470.345,A -85,B 0,C 180,E1 -4800.855,E2 -4800.855} C_VEL
LIN {X 0,Y 523.961,Z 470.345,A -85,B 0,C 180,E1 -4803.735,E2 -4803.735} C_VEL
LIN {X 0,Y 523.906,Z 470.348,A -85,B 0,C 180,E1 -4806.401,E2 -4806.401} C_VEL
LIN {X 0,Y 523.923,Z 470.351,A -85,B 0,C 180,E1 -4809.085,E2 -4809.085} C_VEL
LIN {X 0,Y 523.956,Z 470.34,A -85,B 0,C 180,E1 -4812.119,E2 -4812.119} C_VEL
LIN {X 0,Y 523.956,Z 470.346,A -85,B 0,C 180,E1 -4815.309,E2 -4815.309} C_VEL
LIN {X 0,Y 523.962,Z 470.344,A -85,B 0,C 180,E1 -4818.69,E2 -4818.69} C_VEL
LIN {X 0,Y 523.923,Z 470.351,A -85,B 0,C 180,E1 -4821.08,E2 -4821.08} C_VEL
LIN {X 0,Y 523.905,Z 470.348,A -85,B 0,C 180,E1 -4823.826,E2 -4823.826} C_VEL
LIN {X 0,Y 523.947,Z 470.348,A -85,B 0,C 180,E1 -4826.636,E2 -4826.636} C_VEL
LIN {X 0,Y 523.96,Z 470.344,A -85,B 0,C 180,E1 -4829.356,E2 -4829.356} C_VEL
LIN {X 0,Y 523.983,Z 470.347,A -85,B 0,C 180,E1 -4832.281,E2 -4832.281} C_VEL
LIN {X 0,Y 523.996,Z 470.388,A -85,B 0,C 180,E1 -4835.167,E2 -4835.167} C_VEL
LIN {X 0,Y 526.033,Z 480.186,A -85,B 0,C 180,E1 -4836.789,E2 -4836.789} C_VEL
LIN {X 0,Y 525.663,Z 495.028,A -85,B 0,C 180,E1 -4839.017,E2 -4839.017} C_VEL
LIN {X 0,Y 525.071,Z 515.712,A -85,B 0,C 180,E1 -4842.07,E2 -4842.07} C_VEL
LIN {X 0,Y 524.603,Z 537.531,A -85,B 0,C 180,E1 -4845.254,E2 -4845.254} C_VEL
LIN {X 0,Y 524.485,Z 541.441,A -85,B 0,C 180,E1 -4845.82,E2 -4845.82} C_VEL
LIN {X 0,Y 526.011,Z 552.698,A -85,B 0,C 180,E1 -4846.059,E2 -4846.059} C_VEL
LIN {X 0,Y 525.457,Z 651.425,A -85,B 0,C 180,E1 -4847.467,E2 -4847.467} C_VEL
LIN {X 0,Y 525.291,Z 664.815,A -85,B 0,C 180,E1 -4847.823,E2 -4847.823} C_VEL
LIN {X 0,Y 525.068,Z 677.712,A -85,B 0,C 180,E1 -4848.333,E2 -4848.333} C_VEL
LIN {X 0,Y 524.906,Z 688.572,A -85,B 0,C 180,E1 -4848.903,E2 -4848.903} C_VEL
LIN {X 0,Y 524.571,Z 698.743,A -85,B 0,C 180,E1 -4849.58,E2 -4849.58} C_VEL
LIN {X 0,Y 524.279,Z 709.354,A -85,B 0,C 180,E1 -4850.451,E2 -4850.451} C_VEL
LIN {X 0,Y 524.073,Z 718.011,A -85,B 0,C 180,E1 -4851.323,E2 -4851.323} C_VEL
LIN {X 0,Y 523.829,Z 725.922,A -85,B 0,C 180,E1 -4852.29,E2 -4852.29} C_VEL
LIN {X 0,Y 523.688,Z 732.61,A -85,B 0,C 180,E1 -4853.265,E2 -4853.265} C_VEL
LIN {X 0,Y 523.616,Z 738.003,A -85,B 0,C 180,E1 -4854.222,E2 -4854.222} C_VEL
LIN {X 0,Y 523.447,Z 743.378,A -85,B 0,C 180,E1 -4855.379,E2 -4855.379} C_VEL
LIN {X 0,Y 523.443,Z 747.519,A -85,B 0,C 180,E1 -4856.536,E2 -4856.536} C_VEL
LIN {X 0,Y 523.355,Z 750.693,A -85,B 0,C 180,E1 -4857.691,E2 -4857.691} C_VEL
LIN {X 0,Y 523.28,Z 752.24,A -85,B 0,C 180,E1 -4858.461,E2 -4858.461} C_VEL
LIN {X 0,Y 523.251,Z 753.373,A -85,B 0,C 180,E1 -4859.23,E2 -4859.23} C_VEL
LIN {X 0,Y 523.248,Z 754.103,A -85,B 0,C 180,E1 -4860,E2 -4860} C_VEL
LIN {X 0,Y 523.274,Z 754.377,A -85,B 0,C 180,E1 -4861.539,E2 -4861.539} C_VEL
LIN {X 0,Y 523.333,Z 753.922,A -85,B 0,C 180,E1 -4862.309,E2 -4862.309} C_VEL
LIN {X 0,Y 523.361,Z 753.069,A -85,B 0,C 180,E1 -4863.079,E2 -4863.079} C_VEL
LIN {X 0,Y 523.409,Z 751.81,A -85,B 0,C 180,E1 -4863.85,E2 -4863.85} C_VEL
LIN {X 0,Y 523.365,Z 749.169,A -85,B 0,C 180,E1 -4865.007,E2 -4865.007} C_VEL
LIN {X 0,Y 523.422,Z 745.444,A -85,B 0,C 180,E1 -4866.166,E2 -4866.166} C_VEL
LIN {X 0,Y 523.494,Z 740.691,A -85,B 0,C 180,E1 -4867.327,E2 -4867.327} C_VEL
LIN {X 0,Y 523.654,Z 734.575,A -85,B 0,C 180,E1 -4868.49,E2 -4868.49} C_VEL
LIN {X 0,Y 523.783,Z 726.983,A -85,B 0,C 180,E1 -4869.655,E2 -4869.655} C_VEL
LIN {X 0,Y 524.034,Z 719.27,A -85,B 0,C 180,E1 -4870.626,E2 -4870.626} C_VEL
LIN {X 0,Y 524.227,Z 709.768,A -85,B 0,C 180,E1 -4871.601,E2 -4871.601} C_VEL
LIN {X 0,Y 524.523,Z 699.192,A -85,B 0,C 180,E1 -4872.477,E2 -4872.477} C_VEL
LIN {X 0,Y 524.856,Z 687.389,A -85,B 0,C 180,E1 -4873.256,E2 -4873.256} C_VEL
LIN {X 0,Y 525.082,Z 675.956,A -85,B 0,C 180,E1 -4873.842,E2 -4873.842} C_VEL
LIN {X 0,Y 525.304,Z 662.893,A -85,B 0,C 180,E1 -4874.33,E2 -4874.33} C_VEL
LIN {X 0,Y 525.479,Z 650.253,A -85,B 0,C 180,E1 -4874.647,E2 -4874.647} C_VEL
LIN {X 0,Y 526.014,Z 551.588,A -85,B 0,C 180,E1 -4876.041,E2 -4876.041} C_VEL
LIN {X 0,Y 524.493,Z 541.544,A -85,B 0,C 180,E1 -4876.251,E2 -4876.251} C_VEL
LIN {X 0,Y 524.948,Z 521.639,A -85,B 0,C 180,E1 -4879.148,E2 -4879.148} C_VEL
LIN {X 0,Y 525.44,Z 502.318,A -85,B 0,C 180,E1 -4881.994,E2 -4881.994} C_VEL
LIN {X 0,Y 526.038,Z 482.653,A -85,B 0,C 180,E1 -4884.935,E2 -4884.935} C_VEL
LIN {X 0,Y 525.814,Z 478.796,A -85,B 0,C 180,E1 -4885.534,E2 -4885.534} C_VEL
LIN {X 0,Y 523.981,Z 470.343,A -85,B 0,C 180,E1 -4886.97,E2 -4886.97} C_VEL
LIN {X 0,Y 523.972,Z 470.345,A -85,B 0,C 180,E1 -4887.95,E2 -4887.95} C_VEL
LIN {X 0,Y 523.304,Z 470.428,A -85,B 0,C 180,E1 -4888.591,E2 -4888.591} C_VEL
LIN {X 0,Y 520.445,Z 470.785,A -85,B 0,C 180,E1 -4889.633,E2 -4889.633} C_VEL
LIN {X 0,Y 518.02,Z 471.085,A -85,B 0,C 180,E1 -4890.472,E2 -4890.472} C_VEL
LIN {X 0,Y 516.968,Z 471.214,A -85,B 0,C 180,E1 -4891.12,E2 -4891.12} C_VEL
LIN {X 0,Y 516.876,Z 471.224,A -85,B 0,C 180,E1 -4891.339,E2 -4891.339} C_VEL
LIN {X 0,Y 516.915,Z 471.221,A -85,B 0,C 180,E1 -4893.967,E2 -4893.967} C_VEL
LIN {X 0,Y 516.881,Z 471.22,A -85,B 0,C 180,E1 -4896.746,E2 -4896.746} C_VEL
LIN {X 0,Y 516.885,Z 471.227,A -85,B 0,C 180,E1 -4899.721,E2 -4899.721} C_VEL
LIN {X 0,Y 516.914,Z 471.222,A -85,B 0,C 180,E1 -4901.775,E2 -4901.775} C_VEL
LIN {X 0,Y 516.897,Z 471.219,A -85,B 0,C 180,E1 -4905.007,E2 -4905.007} C_VEL
LIN {X 0,Y 516.918,Z 471.215,A -85,B 0,C 180,E1 -4908.398,E2 -4908.398} C_VEL
LIN {X 0,Y 516.883,Z 471.224,A -85,B 0,C 180,E1 -4911.284,E2 -4911.284} C_VEL
LIN {X 0,Y 516.873,Z 471.222,A -85,B 0,C 180,E1 -4914.22,E2 -4914.22} C_VEL
LIN {X 0,Y 516.897,Z 471.22,A -85,B 0,C 180,E1 -4917.053,E2 -4917.053} C_VEL
LIN {X 0,Y 516.894,Z 471.223,A -85,B 0,C 180,E1 -4919.796,E2 -4919.796} C_VEL
LIN {X 0,Y 516.928,Z 471.214,A -85,B 0,C 180,E1 -4922.467,E2 -4922.467} C_VEL
LIN {X 0,Y 516.911,Z 471.219,A -85,B 0,C 180,E1 -4925.072,E2 -4925.072} C_VEL
LIN {X 0,Y 516.888,Z 471.219,A -85,B 0,C 180,E1 -4928.462,E2 -4928.462} C_VEL
LIN {X 0,Y 516.906,Z 471.218,A -85,B 0,C 180,E1 -4930.955,E2 -4930.955} C_VEL
LIN {X 0,Y 516.917,Z 471.223,A -85,B 0,C 180,E1 -4933.41,E2 -4933.41} C_VEL
LIN {X 0,Y 516.909,Z 471.22,A -85,B 0,C 180,E1 -4935.834,E2 -4935.834} C_VEL
LIN {X 0,Y 516.954,Z 471.213,A -85,B 0,C 180,E1 -4939.028,E2 -4939.028} C_VEL
LIN {X 0,Y 516.982,Z 471.208,A -85,B 0,C 180,E1 -4942.187,E2 -4942.187} C_VEL
LIN {X 0,Y 517.032,Z 471.201,A -85,B 0,C 180,E1 -4944.54,E2 -4944.54} C_VEL
LIN {X 0,Y 517.088,Z 471.2,A -85,B 0,C 180,E1 -4947.663,E2 -4947.663} C_VEL
LIN {X 0,Y 517.095,Z 471.194,A -85,B 0,C 180,E1 -4950.779,E2 -4950.779} C_VEL
LIN {X 0,Y 517.016,Z 471.207,A -85,B 0,C 180,E1 -4953.117,E2 -4953.117} C_VEL
LIN {X 0,Y 517.005,Z 471.204,A -85,B 0,C 180,E1 -4956.243,E2 -4956.243} C_VEL
LIN {X 0,Y 516.954,Z 471.22,A -85,B 0,C 180,E1 -4959.389,E2 -4959.389} C_VEL
LIN {X 0,Y 516.954,Z 471.214,A -85,B 0,C 180,E1 -4961.807,E2 -4961.807} C_VEL
LIN {X 0,Y 516.947,Z 471.217,A -85,B 0,C 180,E1 -4965.147,E2 -4965.147} C_VEL
LIN {X 0,Y 516.927,Z 471.214,A -85,B 0,C 180,E1 -4968.222,E2 -4968.222} C_VEL
LIN {X 0,Y 516.915,Z 471.216,A -85,B 0,C 180,E1 -4970.701,E2 -4970.701} C_VEL
LIN {X 0,Y 516.914,Z 471.216,A -85,B 0,C 180,E1 -4974.072,E2 -4974.072} C_VEL
LIN {X 0,Y 516.928,Z 471.215,A -85,B 0,C 180,E1 -4976.658,E2 -4976.658} C_VEL
LIN {X 0,Y 516.913,Z 471.222,A -85,B 0,C 180,E1 -4979.524,E2 -4979.524} C_VEL
LIN {X 0,Y 516.897,Z 471.218,A -85,B 0,C 180,E1 -4982.543,E2 -4982.543} C_VEL
LIN {X 0,Y 516.868,Z 471.231,A -85,B 0,C 180,E1 -4985.33,E2 -4985.33} C_VEL
LIN {X 0,Y 516.883,Z 471.221,A -85,B 0,C 180,E1 -4987.943,E2 -4987.943} C_VEL
LIN {X 0,Y 516.888,Z 471.22,A -85,B 0,C 180,E1 -4990.741,E2 -4990.741} C_VEL
LIN {X 0,Y 516.907,Z 471.219,A -85,B 0,C 180,E1 -4992.829,E2 -4992.829} C_VEL
LIN {X 0,Y 516.925,Z 471.219,A -85,B 0,C 180,E1 -4995.01,E2 -4995.01} C_VEL
LIN {X 0,Y 516.915,Z 471.215,A -85,B 0,C 180,E1 -4998.399,E2 -4998.399} C_VEL
LIN {X 0,Y 516.884,Z 471.229,A -85,B 0,C 180,E1 -5001.284,E2 -5001.284} C_VEL
LIN {X 0,Y 516.875,Z 471.22,A -85,B 0,C 180,E1 -5004.22,E2 -5004.22} C_VEL
LIN {X 0,Y 516.897,Z 471.223,A -85,B 0,C 180,E1 -5007.053,E2 -5007.053} C_VEL
LIN {X 0,Y 516.895,Z 471.221,A -85,B 0,C 180,E1 -5009.796,E2 -5009.796} C_VEL
LIN {X 0,Y 516.929,Z 471.216,A -85,B 0,C 180,E1 -5012.467,E2 -5012.467} C_VEL
LIN {X 0,Y 516.992,Z 471.388,A -85,B 0,C 180,E1 -5014.049,E2 -5014.049} C_VEL
LIN {X 0,Y 518.978,Z 481.622,A -85,B 0,C 180,E1 -5015.618,E2 -5015.618} C_VEL
LIN {X 0,Y 518.61,Z 499.085,A -85,B 0,C 180,E1 -5018.12,E2 -5018.12} C_VEL
LIN {X 0,Y 518.106,Z 520.831,A -85,B 0,C 180,E1 -5021.227,E2 -5021.227} C_VEL
LIN {X 0,Y 517.632,Z 541.95,A -85,B 0,C 180,E1 -5024.244,E2 -5024.244} C_VEL
LIN {X 0,Y 517.572,Z 545.04,A -85,B 0,C 180,E1 -5024.682,E2 -5024.682} C_VEL
LIN {X 0,Y 519.074,Z 556.089,A -85,B 0,C 180,E1 -5024.902,E2 -5024.902} C_VEL
LIN {X 0,Y 518.565,Z 654.097,A -85,B 0,C 180,E1 -5026.305,E2 -5026.305} C_VEL
LIN {X 0,Y 518.391,Z 666.609,A -85,B 0,C 180,E1 -5026.625,E2 -5026.625} C_VEL
LIN {X 0,Y 518.132,Z 679.407,A -85,B 0,C 180,E1 -5027.117,E2 -5027.117} C_VEL
LIN {X 0,Y 517.84,Z 691.223,A -85,B 0,C 180,E1 -5027.734,E2 -5027.734} C_VEL
LIN {X 0,Y 517.596,Z 701.932,A -85,B 0,C 180,E1 -5028.447,E2 -5028.447} C_VEL
LIN {X 0,Y 517.252,Z 712.551,A -85,B 0,C 180,E1 -5029.332,E2 -5029.332} C_VEL
LIN {X 0,Y 517.063,Z 721.199,A -85,B 0,C 180,E1 -5030.218,E2 -5030.218} C_VEL
LIN {X 0,Y 516.82,Z 729.159,A -85,B 0,C 180,E1 -5031.2,E2 -5031.2} C_VEL
LIN {X 0,Y 516.623,Z 735.754,A -85,B 0,C 180,E1 -5032.181,E2 -5032.181} C_VEL
LIN {X 0,Y 516.491,Z 741.365,A -85,B 0,C 180,E1 -5033.186,E2 -5033.186} C_VEL
LIN {X 0,Y 516.471,Z 745.792,A -85,B 0,C 180,E1 -5034.142,E2 -5034.142} C_VEL
LIN {X 0,Y 516.278,Z 750.146,A -85,B 0,C 180,E1 -5035.315,E2 -5035.315} C_VEL
LIN {X 0,Y 516.373,Z 752.493,A -85,B 0,C 180,E1 -5036.098,E2 -5036.098} C_VEL
LIN {X 0,Y 516.283,Z 754.332,A -85,B 0,C 180,E1 -5036.879,E2 -5036.879} C_VEL
LIN {X 0,Y 516.192,Z 756.795,A -85,B 0,C 180,E1 -5038.44,E2 -5038.44} C_VEL
LIN {X 0,Y 516.16,Z 757.403,A -85,B 0,C 180,E1 -5039.22,E2 -5039.22} C_VEL
LIN {X 0,Y 516.16,Z 757.458,A -85,B 0,C 180,E1 -5040.78,E2 -5040.78} C_VEL
LIN {X 0,Y 516.192,Z 756.886,A -85,B 0,C 180,E1 -5041.56,E2 -5041.56} C_VEL
LIN {X 0,Y 516.283,Z 754.541,A -85,B 0,C 180,E1 -5043.121,E2 -5043.121} C_VEL
LIN {X 0,Y 516.36,Z 751.666,A -85,B 0,C 180,E1 -5044.293,E2 -5044.293} C_VEL
LIN {X 0,Y 516.4,Z 747.753,A -85,B 0,C 180,E1 -5045.467,E2 -5045.467} C_VEL
LIN {X 0,Y 516.462,Z 742.932,A -85,B 0,C 180,E1 -5046.593,E2 -5046.593} C_VEL
LIN {X 0,Y 516.619,Z 736.316,A -85,B 0,C 180,E1 -5047.819,E2 -5047.819} C_VEL
LIN {X 0,Y 516.791,Z 728.386,A -85,B 0,C 180,E1 -5048.998,E2 -5048.998} C_VEL
LIN {X 0,Y 517.046,Z 720.266,A -85,B 0,C 180,E1 -5049.98,E2 -5049.98} C_VEL
LIN {X 0,Y 517.336,Z 710.258,A -85,B 0,C 180,E1 -5050.964,E2 -5050.964} C_VEL
LIN {X 0,Y 517.615,Z 699.377,A -85,B 0,C 180,E1 -5051.825,E2 -5051.825} C_VEL
LIN {X 0,Y 517.906,Z 687.974,A -85,B 0,C 180,E1 -5052.54,E2 -5052.54} C_VEL
LIN {X 0,Y 518.188,Z 675.534,A -85,B 0,C 180,E1 -5053.131,E2 -5053.131} C_VEL
LIN {X 0,Y 518.418,Z 662.624,A -85,B 0,C 180,E1 -5053.574,E2 -5053.574} C_VEL
LIN {X 0,Y 518.566,Z 650.141,A -85,B 0,C 180,E1 -5053.845,E2 -5053.845} C_VEL
LIN {X 0,Y 518.99,Z 554.38,A -85,B 0,C 180,E1 -5055.218,E2 -5055.218} C_VEL
LIN {X 0,Y 517.575,Z 545.015,A -85,B 0,C 180,E1 -5055.423,E2 -5055.423} C_VEL
LIN {X 0,Y 517.92,Z 528.385,A -85,B 0,C 180,E1 -5057.777,E2 -5057.777} C_VEL
LIN {X 0,Y 518.18,Z 515.389,A -85,B 0,C 180,E1 -5059.614,E2 -5059.614} C_VEL
LIN {X 0,Y 518.514,Z 494.747,A -85,B 0,C 180,E1 -5062.441,E2 -5062.441} C_VEL
LIN {X 0,Y 518.691,Z 480.544,A -85,B 0,C 180,E1 -5064.367,E2 -5064.367} C_VEL
LIN {X 0,Y 516.947,Z 471.218,A -85,B 0,C 180,E1 -5065.734,E2 -5065.734} C_VEL
LIN {X 0,Y 516.921,Z 471.223,A -85,B 0,C 180,E1 -5068.415,E2 -5068.415} C_VEL
LIN {X 0,Y 516.892,Z 471.226,A -85,B 0,C 180,E1 -5071.109,E2 -5071.109} C_VEL
LIN {X 0,Y 516.911,Z 471.22,A -85,B 0,C 180,E1 -5073.966,E2 -5073.966} C_VEL
LIN {X 0,Y 516.879,Z 471.228,A -85,B 0,C 180,E1 -5076.746,E2 -5076.746} C_VEL
LIN {X 0,Y 516.885,Z 471.221,A -85,B 0,C 180,E1 -5079.721,E2 -5079.721} C_VEL
LIN {X 0,Y 516.914,Z 471.217,A -85,B 0,C 180,E1 -5081.775,E2 -5081.775} C_VEL
LIN {X 0,Y 516.925,Z 471.217,A -85,B 0,C 180,E1 -5085.01,E2 -5085.01} C_VEL
LIN {X 0,Y 516.918,Z 471.224,A -85,B 0,C 180,E1 -5088.398,E2 -5088.398} C_VEL
LIN {X 0,Y 516.883,Z 471.221,A -85,B 0,C 180,E1 -5091.284,E2 -5091.284} C_VEL
LIN {X 0,Y 516.892,Z 471.226,A -85,B 0,C 180,E1 -5094.221,E2 -5094.221} C_VEL
LIN {X 0,Y 516.9,Z 471.22,A -85,B 0,C 180,E1 -5097.053,E2 -5097.053} C_VEL
LIN {X 0,Y 516.904,Z 471.222,A -85,B 0,C 180,E1 -5099.797,E2 -5099.797} C_VEL
LIN {X 0,Y 516.93,Z 471.223,A -85,B 0,C 180,E1 -5102.467,E2 -5102.467} C_VEL
LIN {X 0,Y 516.955,Z 471.259,A -85,B 0,C 180,E1 -5104.401,E2 -5104.401} C_VEL
LIN {X 0,Y 519.549,Z 482.593,A -85,B 0,C 180,E1 -5106.058,E2 -5106.058} C_VEL
LIN {X 0,Y 519.524,Z 489.035,A -85,B 0,C 180,E1 -5106.91,E2 -5106.91} C_VEL
LIN {X 0,Y 518.682,Z 514.489,A -85,B 0,C 180,E1 -5110.2,E2 -5110.2} C_VEL
LIN {X 0,Y 518.41,Z 524.353,A -85,B 0,C 180,E1 -5111.456,E2 -5111.456} C_VEL
LIN {X 0,Y 520.275,Z 536.259,A -85,B 0,C 180,E1 -5111.703,E2 -5111.703} C_VEL
LIN {X 0,Y 519.516,Z 656.529,A -85,B 0,C 180,E1 -5113.395,E2 -5113.395} C_VEL
LIN {X 0,Y 519.319,Z 670.596,A -85,B 0,C 180,E1 -5113.681,E2 -5113.681} C_VEL
LIN {X 0,Y 519.077,Z 684.474,A -85,B 0,C 180,E1 -5114.12,E2 -5114.12} C_VEL
LIN {X 0,Y 518.739,Z 698.474,A -85,B 0,C 180,E1 -5114.731,E2 -5114.731} C_VEL
LIN {X 0,Y 518.302,Z 711.53,A -85,B 0,C 180,E1 -5115.472,E2 -5115.472} C_VEL
LIN {X 0,Y 517.906,Z 724.038,A -85,B 0,C 180,E1 -5116.362,E2 -5116.362} C_VEL
LIN {X 0,Y 517.543,Z 735.325,A -85,B 0,C 180,E1 -5117.351,E2 -5117.351} C_VEL
LIN {X 0,Y 517.232,Z 745.568,A -85,B 0,C 180,E1 -5118.439,E2 -5118.439} C_VEL
LIN {X 0,Y 516.935,Z 754.831,A -85,B 0,C 180,E1 -5119.622,E2 -5119.622} C_VEL
LIN {X 0,Y 516.667,Z 763.665,A -85,B 0,C 180,E1 -5121,E2 -5121} C_VEL
LIN {X 0,Y 516.501,Z 769.881,A -85,B 0,C 180,E1 -5122.18,E2 -5122.18} C_VEL
LIN {X 0,Y 516.396,Z 776.471,A -85,B 0,C 180,E1 -5123.749,E2 -5123.749} C_VEL
LIN {X 0,Y 516.305,Z 780.322,A -85,B 0,C 180,E1 -5124.924,E2 -5124.924} C_VEL
LIN {X 0,Y 516.325,Z 783.288,A -85,B 0,C 180,E1 -5126.098,E2 -5126.098} C_VEL
LIN {X 0,Y 516.258,Z 785.997,A -85,B 0,C 180,E1 -5127.659,E2 -5127.659} C_VEL
LIN {X 0,Y 516.157,Z 787.333,A -85,B 0,C 180,E1 -5129.22,E2 -5129.22} C_VEL
LIN {X 0,Y 516.157,Z 787.333,A -85,B 0,C 180,E1 -5130.78,E2 -5130.78} C_VEL
LIN {X 0,Y 516.258,Z 786,A -85,B 0,C 180,E1 -5132.341,E2 -5132.341} C_VEL
LIN {X 0,Y 516.325,Z 783.292,A -85,B 0,C 180,E1 -5133.903,E2 -5133.903} C_VEL
LIN {X 0,Y 516.388,Z 779.128,A -85,B 0,C 180,E1 -5135.467,E2 -5135.467} C_VEL
LIN {X 0,Y 516.403,Z 773.38,A -85,B 0,C 180,E1 -5137.036,E2 -5137.036} C_VEL
LIN {X 0,Y 516.599,Z 766.893,A -85,B 0,C 180,E1 -5138.41,E2 -5138.41} C_VEL
LIN {X 0,Y 516.801,Z 758.814,A -85,B 0,C 180,E1 -5139.787,E2 -5139.787} C_VEL
LIN {X 0,Y 517.069,Z 750.341,A -85,B 0,C 180,E1 -5140.97,E2 -5140.97} C_VEL
LIN {X 0,Y 517.41,Z 739.747,A -85,B 0,C 180,E1 -5142.191,E2 -5142.191} C_VEL
LIN {X 0,Y 517.758,Z 728.603,A -85,B 0,C 180,E1 -5143.242,E2 -5143.242} C_VEL
LIN {X 0,Y 518.108,Z 717.127,A -85,B 0,C 180,E1 -5144.133,E2 -5144.133} C_VEL
LIN {X 0,Y 518.553,Z 704.55,A -85,B 0,C 180,E1 -5144.922,E2 -5144.922} C_VEL
LIN {X 0,Y 518.878,Z 690.436,A -85,B 0,C 180,E1 -5145.617,E2 -5145.617} C_VEL
LIN {X 0,Y 519.186,Z 676.61,A -85,B 0,C 180,E1 -5146.121,E2 -5146.121} C_VEL
LIN {X 0,Y 519.445,Z 661.978,A -85,B 0,C 180,E1 -5146.485,E2 -5146.485} C_VEL
LIN {X 0,Y 520.177,Z 535.983,A -85,B 0,C 180,E1 -5148.277,E2 -5148.277} C_VEL
LIN {X 0,Y 518.393,Z 524.366,A -85,B 0,C 180,E1 -5148.519,E2 -5148.519} C_VEL
LIN {X 0,Y 519.184,Z 498.472,A -85,B 0,C 180,E1 -5151.855,E2 -5151.855} C_VEL
LIN {X 0,Y 519.758,Z 484.33,A -85,B 0,C 180,E1 -5153.72,E2 -5153.72} C_VEL
LIN {X 0,Y 517.86,Z 475.08,A -85,B 0,C 180,E1 -5155.094,E2 -5155.094} C_VEL
LIN {X 0,Y 516.937,Z 471.222,A -85,B 0,C 180,E1 -5155.708,E2 -5155.708} C_VEL
LIN {X 0,Y 516.922,Z 471.221,A -85,B 0,C 180,E1 -5158.415,E2 -5158.415} C_VEL
LIN {X 0,Y 516.893,Z 471.227,A -85,B 0,C 180,E1 -5161.109,E2 -5161.109} C_VEL
LIN {X 0,Y 516.91,Z 471.222,A -85,B 0,C 180,E1 -5163.966,E2 -5163.966} C_VEL
LIN {X 0,Y 516.879,Z 471.225,A -85,B 0,C 180,E1 -5166.746,E2 -5166.746} C_VEL
LIN {X 0,Y 516.885,Z 471.225,A -85,B 0,C 180,E1 -5169.721,E2 -5169.721} C_VEL
LIN {X 0,Y 516.909,Z 471.221,A -85,B 0,C 180,E1 -5172.761,E2 -5172.761} C_VEL
LIN {X 0,Y 516.926,Z 471.222,A -85,B 0,C 180,E1 -5175.01,E2 -5175.01} C_VEL
LIN {X 0,Y 516.918,Z 471.219,A -85,B 0,C 180,E1 -5178.399,E2 -5178.399} C_VEL
LIN {X 0,Y 516.886,Z 471.226,A -85,B 0,C 180,E1 -5181.284,E2 -5181.284} C_VEL
LIN {X 0,Y 516.877,Z 471.225,A -85,B 0,C 180,E1 -5184.22,E2 -5184.22} C_VEL
LIN {X 0,Y 516.9,Z 471.226,A -85,B 0,C 180,E1 -5187.053,E2 -5187.053} C_VEL
LIN {X 0,Y 516.896,Z 471.223,A -85,B 0,C 180,E1 -5189.797,E2 -5189.797} C_VEL
LIN {X 0,Y 516.932,Z 471.226,A -85,B 0,C 180,E1 -5192.468,E2 -5192.468} C_VEL
LIN {X 0,Y 516.944,Z 471.337,A -85,B 0,C 180,E1 -5194.912,E2 -5194.912} C_VEL
LIN {X 0,Y 519.162,Z 481.732,A -85,B 0,C 180,E1 -5196.674,E2 -5196.674} C_VEL
LIN {X 0,Y 518.822,Z 495.327,A -85,B 0,C 180,E1 -5198.753,E2 -5198.753} C_VEL
LIN {X 0,Y 518.166,Z 515.814,A -85,B 0,C 180,E1 -5201.823,E2 -5201.823} C_VEL
LIN {X 0,Y 517.653,Z 537.655,A -85,B 0,C 180,E1 -5205.051,E2 -5205.051} C_VEL
LIN {X 0,Y 517.543,Z 541.406,A -85,B 0,C 180,E1 -5205.601,E2 -5205.601} C_VEL
LIN {X 0,Y 519.211,Z 553.604,A -85,B 0,C 180,E1 -5205.848,E2 -5205.848} C_VEL
LIN {X 0,Y 518.556,Z 651.682,A -85,B 0,C 180,E1 -5207.297,E2 -5207.297} C_VEL
LIN {X 0,Y 518.373,Z 665.051,A -85,B 0,C 180,E1 -5207.66,E2 -5207.66} C_VEL
LIN {X 0,Y 518.125,Z 677.965,A -85,B 0,C 180,E1 -5208.177,E2 -5208.177} C_VEL
LIN {X 0,Y 517.888,Z 690.305,A -85,B 0,C 180,E1 -5208.85,E2 -5208.85} C_VEL
LIN {X 0,Y 517.484,Z 701.531,A -85,B 0,C 180,E1 -5209.633,E2 -5209.633} C_VEL
LIN {X 0,Y 517.206,Z 711.61,A -85,B 0,C 180,E1 -5210.517,E2 -5210.517} C_VEL
LIN {X 0,Y 516.931,Z 721.546,A -85,B 0,C 180,E1 -5211.596,E2 -5211.596} C_VEL
LIN {X 0,Y 516.696,Z 730.255,A -85,B 0,C 180,E1 -5212.772,E2 -5212.772} C_VEL
LIN {X 0,Y 516.612,Z 737.246,A -85,B 0,C 180,E1 -5213.948,E2 -5213.948} C_VEL
LIN {X 0,Y 516.362,Z 743.616,A -85,B 0,C 180,E1 -5215.316,E2 -5215.316} C_VEL
LIN {X 0,Y 516.357,Z 747.774,A -85,B 0,C 180,E1 -5216.489,E2 -5216.489} C_VEL
LIN {X 0,Y 516.282,Z 750.926,A -85,B 0,C 180,E1 -5217.659,E2 -5217.659} C_VEL
LIN {X 0,Y 516.197,Z 752.464,A -85,B 0,C 180,E1 -5218.44,E2 -5218.44} C_VEL
LIN {X 0,Y 516.161,Z 753.59,A -85,B 0,C 180,E1 -5219.22,E2 -5219.22} C_VEL
LIN {X 0,Y 516.155,Z 754.31,A -85,B 0,C 180,E1 -5220,E2 -5220} C_VEL
LIN {X 0,Y 516.192,Z 754.561,A -85,B 0,C 180,E1 -5221.56,E2 -5221.56} C_VEL
LIN {X 0,Y 516.259,Z 754.099,A -85,B 0,C 180,E1 -5222.341,E2 -5222.341} C_VEL
LIN {X 0,Y 516.275,Z 753.238,A -85,B 0,C 180,E1 -5223.121,E2 -5223.121} C_VEL
LIN {X 0,Y 516.332,Z 751.966,A -85,B 0,C 180,E1 -5223.902,E2 -5223.902} C_VEL
LIN {X 0,Y 516.295,Z 749.314,A -85,B 0,C 180,E1 -5225.076,E2 -5225.076} C_VEL
LIN {X 0,Y 516.331,Z 745.568,A -85,B 0,C 180,E1 -5226.251,E2 -5226.251} C_VEL
LIN {X 0,Y 516.436,Z 740.764,A -85,B 0,C 180,E1 -5227.428,E2 -5227.428} C_VEL
LIN {X 0,Y 516.601,Z 734.625,A -85,B 0,C 180,E1 -5228.606,E2 -5228.606} C_VEL
LIN {X 0,Y 516.75,Z 726.975,A -85,B 0,C 180,E1 -5229.788,E2 -5229.788} C_VEL
LIN {X 0,Y 517.024,Z 719.2,A -85,B 0,C 180,E1 -5230.772,E2 -5230.772} C_VEL
LIN {X 0,Y 517.198,Z 709.653,A -85,B 0,C 180,E1 -5231.761,E2 -5231.761} C_VEL
LIN {X 0,Y 517.555,Z 698.985,A -85,B 0,C 180,E1 -5232.648,E2 -5232.648} C_VEL
LIN {X 0,Y 517.926,Z 687.064,A -85,B 0,C 180,E1 -5233.437,E2 -5233.437} C_VEL
LIN {X 0,Y 518.168,Z 675.509,A -85,B 0,C 180,E1 -5234.031,E2 -5234.031} C_VEL
LIN {X 0,Y 518.389,Z 662.263,A -85,B 0,C 180,E1 -5234.526,E2 -5234.526} C_VEL
LIN {X 0,Y 518.593,Z 649.087,A -85,B 0,C 180,E1 -5234.846,E2 -5234.846} C_VEL
LIN {X 0,Y 519.108,Z 551.786,A -85,B 0,C 180,E1 -5236.251,E2 -5236.251} C_VEL
LIN {X 0,Y 517.512,Z 541.499,A -85,B 0,C 180,E1 -5236.47,E2 -5236.47} C_VEL
LIN {X 0,Y 518.001,Z 522.914,A -85,B 0,C 180,E1 -5239.209,E2 -5239.209} C_VEL
LIN {X 0,Y 518.512,Z 503.585,A -85,B 0,C 180,E1 -5242.094,E2 -5242.094} C_VEL
LIN {X 0,Y 519.137,Z 485.035,A -85,B 0,C 180,E1 -5244.9,E2 -5244.9} C_VEL
LIN {X 0,Y 518.854,Z 480.048,A -85,B 0,C 180,E1 -5245.687,E2 -5245.687} C_VEL
LIN {X 0,Y 516.943,Z 471.221,A -85,B 0,C 180,E1 -5247.203,E2 -5247.203} C_VEL
LIN {X 0,Y 516.895,Z 471.223,A -85,B 0,C 180,E1 -5250.204,E2 -5250.204} C_VEL
LIN {X 0,Y 516.876,Z 471.224,A -85,B 0,C 180,E1 -5251.339,E2 -5251.339} C_VEL
LIN {X 0,Y 516.196,Z 471.311,A -85,B 0,C 180,E1 -5251.99,E2 -5251.99} C_VEL
LIN {X 0,Y 513.352,Z 471.663,A -85,B 0,C 180,E1 -5253.047,E2 -5253.047} C_VEL
LIN {X 0,Y 510.954,Z 471.965,A -85,B 0,C 180,E1 -5253.898,E2 -5253.898} C_VEL
LIN {X 0,Y 509.919,Z 472.089,A -85,B 0,C 180,E1 -5254.555,E2 -5254.555} C_VEL
LIN {X 0,Y 509.832,Z 472.099,A -85,B 0,C 180,E1 -5254.777,E2 -5254.777} C_VEL
LIN {X 0,Y 509.82,Z 472.105,A -85,B 0,C 180,E1 -5257.341,E2 -5257.341} C_VEL
LIN {X 0,Y 509.841,Z 472.097,A -85,B 0,C 180,E1 -5260.382,E2 -5260.382} C_VEL
LIN {X 0,Y 509.825,Z 472.101,A -85,B 0,C 180,E1 -5263.062,E2 -5263.062} C_VEL
LIN {X 0,Y 509.826,Z 472.104,A -85,B 0,C 180,E1 -5265.793,E2 -5265.793} C_VEL
LIN {X 0,Y 509.859,Z 472.094,A -85,B 0,C 180,E1 -5268.574,E2 -5268.574} C_VEL
LIN {X 0,Y 509.853,Z 472.101,A -85,B 0,C 180,E1 -5271.786,E2 -5271.786} C_VEL
LIN {X 0,Y 509.832,Z 472.098,A -85,B 0,C 180,E1 -5274.622,E2 -5274.622} C_VEL
LIN {X 0,Y 509.863,Z 472.102,A -85,B 0,C 180,E1 -5277.481,E2 -5277.481} C_VEL
LIN {X 0,Y 509.861,Z 472.095,A -85,B 0,C 180,E1 -5280.274,E2 -5280.274} C_VEL
LIN {X 0,Y 509.886,Z 472.093,A -85,B 0,C 180,E1 -5282.944,E2 -5282.944} C_VEL
LIN {X 0,Y 509.866,Z 472.102,A -85,B 0,C 180,E1 -5285.574,E2 -5285.574} C_VEL
LIN {X 0,Y 509.853,Z 472.097,A -85,B 0,C 180,E1 -5288.998,E2 -5288.998} C_VEL
LIN {X 0,Y 509.891,Z 472.093,A -85,B 0,C 180,E1 -5291.999,E2 -5291.999} C_VEL
LIN {X 0,Y 509.913,Z 472.089,A -85,B 0,C 180,E1 -5294.819,E2 -5294.819} C_VEL
LIN {X 0,Y 509.903,Z 472.09,A -85,B 0,C 180,E1 -5298.124,E2 -5298.124} C_VEL
LIN {X 0,Y 509.921,Z 472.093,A -85,B 0,C 180,E1 -5301.28,E2 -5301.28} C_VEL
LIN {X 0,Y 509.981,Z 472.085,A -85,B 0,C 180,E1 -5303.67,E2 -5303.67} C_VEL
LIN {X 0,Y 510.058,Z 472.076,A -85,B 0,C 180,E1 -5307.631,E2 -5307.631} C_VEL
LIN {X 0,Y 510.066,Z 472.07,A -85,B 0,C 180,E1 -5310.789,E2 -5310.789} C_VEL
LIN {X 0,Y 509.959,Z 472.087,A -85,B 0,C 180,E1 -5313.16,E2 -5313.16} C_VEL
LIN {X 0,Y 509.956,Z 472.082,A -85,B 0,C 180,E1 -5316.33,E2 -5316.33} C_VEL
LIN {X 0,Y 509.917,Z 472.088,A -85,B 0,C 180,E1 -5318.72,E2 -5318.72} C_VEL
LIN {X 0,Y 509.906,Z 472.091,A -85,B 0,C 180,E1 -5321.932,E2 -5321.932} C_VEL
LIN {X 0,Y 509.896,Z 472.097,A -85,B 0,C 180,E1 -5325.242,E2 -5325.242} C_VEL
LIN {X 0,Y 509.89,Z 472.092,A -85,B 0,C 180,E1 -5328.001,E2 -5328.001} C_VEL
LIN {X 0,Y 509.853,Z 472.099,A -85,B 0,C 180,E1 -5331.002,E2 -5331.002} C_VEL
LIN {X 0,Y 509.839,Z 472.103,A -85,B 0,C 180,E1 -5333.563,E2 -5333.563} C_VEL
LIN {X 0,Y 509.914,Z 472.088,A -85,B 0,C 180,E1 -5336.379,E2 -5336.379} C_VEL
LIN {X 0,Y 509.879,Z 472.094,A -85,B 0,C 180,E1 -5338.844,E2 -5338.844} C_VEL
LIN {X 0,Y 509.822,Z 472.104,A -85,B 0,C 180,E1 -5341.59,E2 -5341.59} C_VEL
LIN {X 0,Y 509.849,Z 472.096,A -85,B 0,C 180,E1 -5344.414,E2 -5344.414} C_VEL
LIN {X 0,Y 509.819,Z 472.109,A -85,B 0,C 180,E1 -5347.341,E2 -5347.341} C_VEL
LIN {X 0,Y 509.841,Z 472.097,A -85,B 0,C 180,E1 -5350.382,E2 -5350.382} C_VEL
LIN {X 0,Y 509.843,Z 472.102,A -85,B 0,C 180,E1 -5353.064,E2 -5353.064} C_VEL
LIN {X 0,Y 509.832,Z 472.1,A -85,B 0,C 180,E1 -5355.792,E2 -5355.792} C_VEL
LIN {X 0,Y 509.857,Z 472.095,A -85,B 0,C 180,E1 -5358.575,E2 -5358.575} C_VEL
LIN {X 0,Y 509.854,Z 472.097,A -85,B 0,C 180,E1 -5361.787,E2 -5361.787} C_VEL
LIN {X 0,Y 509.835,Z 472.099,A -85,B 0,C 180,E1 -5364.622,E2 -5364.622} C_VEL
LIN {X 0,Y 509.864,Z 472.1,A -85,B 0,C 180,E1 -5367.481,E2 -5367.481} C_VEL
LIN {X 0,Y 509.861,Z 472.095,A -85,B 0,C 180,E1 -5370.274,E2 -5370.274} C_VEL
LIN {X 0,Y 509.887,Z 472.097,A -85,B 0,C 180,E1 -5372.944,E2 -5372.944} C_VEL
LIN {X 0,Y 509.913,Z 472.139,A -85,B 0,C 180,E1 -5373.829,E2 -5373.829} C_VEL
LIN {X 0,Y 512.083,Z 483.076,A -85,B 0,C 180,E1 -5375.524,E2 -5375.524} C_VEL
LIN {X 0,Y 511.693,Z 500.348,A -85,B 0,C 180,E1 -5378.021,E2 -5378.021} C_VEL
LIN {X 0,Y 511.214,Z 520.65,A -85,B 0,C 180,E1 -5380.943,E2 -5380.943} C_VEL
LIN {X 0,Y 510.656,Z 543.987,A -85,B 0,C 180,E1 -5384.295,E2 -5384.295} C_VEL
LIN {X 0,Y 510.615,Z 545.271,A -85,B 0,C 180,E1 -5384.479,E2 -5384.479} C_VEL
LIN {X 0,Y 512.212,Z 556.412,A -85,B 0,C 180,E1 -5384.701,E2 -5384.701} C_VEL
LIN {X 0,Y 511.649,Z 654.569,A -85,B 0,C 180,E1 -5386.142,E2 -5386.142} C_VEL
LIN {X 0,Y 511.441,Z 667.732,A -85,B 0,C 180,E1 -5386.491,E2 -5386.491} C_VEL
LIN {X 0,Y 511.178,Z 680.213,A -85,B 0,C 180,E1 -5386.989,E2 -5386.989} C_VEL
LIN {X 0,Y 510.861,Z 692.08,A -85,B 0,C 180,E1 -5387.624,E2 -5387.624} C_VEL
LIN {X 0,Y 510.585,Z 703.167,A -85,B 0,C 180,E1 -5388.387,E2 -5388.387} C_VEL
LIN {X 0,Y 510.213,Z 713.553,A -85,B 0,C 180,E1 -5389.283,E2 -5389.283} C_VEL
LIN {X 0,Y 509.978,Z 722.951,A -85,B 0,C 180,E1 -5390.281,E2 -5390.281} C_VEL
LIN {X 0,Y 509.731,Z 730.67,A -85,B 0,C 180,E1 -5391.277,E2 -5391.277} C_VEL
LIN {X 0,Y 509.503,Z 738.201,A -85,B 0,C 180,E1 -5392.47,E2 -5392.47} C_VEL
LIN {X 0,Y 509.367,Z 744.227,A -85,B 0,C 180,E1 -5393.663,E2 -5393.663} C_VEL
LIN {X 0,Y 509.252,Z 748.995,A -85,B 0,C 180,E1 -5394.853,E2 -5394.853} C_VEL
LIN {X 0,Y 509.304,Z 752.643,A -85,B 0,C 180,E1 -5396.044,E2 -5396.044} C_VEL
LIN {X 0,Y 509.202,Z 754.512,A -85,B 0,C 180,E1 -5396.835,E2 -5396.835} C_VEL
LIN {X 0,Y 509.189,Z 755.945,A -85,B 0,C 180,E1 -5397.627,E2 -5397.627} C_VEL
LIN {X 0,Y 509.113,Z 756.973,A -85,B 0,C 180,E1 -5398.418,E2 -5398.418} C_VEL
LIN {X 0,Y 509.065,Z 757.822,A -85,B 0,C 180,E1 -5400,E2 -5400} C_VEL
LIN {X 0,Y 509.074,Z 757.652,A -85,B 0,C 180,E1 -5400.791,E2 -5400.791} C_VEL
LIN {X 0,Y 509.189,Z 756.097,A -85,B 0,C 180,E1 -5402.373,E2 -5402.373} C_VEL
LIN {X 0,Y 509.202,Z 754.728,A -85,B 0,C 180,E1 -5403.165,E2 -5403.165} C_VEL
LIN {X 0,Y 509.281,Z 751.846,A -85,B 0,C 180,E1 -5404.353,E2 -5404.353} C_VEL
LIN {X 0,Y 509.34,Z 747.924,A -85,B 0,C 180,E1 -5405.543,E2 -5405.543} C_VEL
LIN {X 0,Y 509.417,Z 742.194,A -85,B 0,C 180,E1 -5406.864,E2 -5406.864} C_VEL
LIN {X 0,Y 509.612,Z 735.217,A -85,B 0,C 180,E1 -5408.126,E2 -5408.126} C_VEL
LIN {X 0,Y 509.83,Z 726.926,A -85,B 0,C 180,E1 -5409.322,E2 -5409.322} C_VEL
LIN {X 0,Y 510.064,Z 718.391,A -85,B 0,C 180,E1 -5410.319,E2 -5410.319} C_VEL
LIN {X 0,Y 510.422,Z 707.903,A -85,B 0,C 180,E1 -5411.315,E2 -5411.315} C_VEL
LIN {X 0,Y 510.754,Z 696.986,A -85,B 0,C 180,E1 -5412.142,E2 -5412.142} C_VEL
LIN {X 0,Y 510.99,Z 685.785,A -85,B 0,C 180,E1 -5412.814,E2 -5412.814} C_VEL
LIN {X 0,Y 511.25,Z 673.866,A -85,B 0,C 180,E1 -5413.363,E2 -5413.363} C_VEL
LIN {X 0,Y 511.504,Z 660.819,A -85,B 0,C 180,E1 -5413.786,E2 -5413.786} C_VEL
LIN {X 0,Y 511.693,Z 646.936,A -85,B 0,C 180,E1 -5414.06,E2 -5414.06} C_VEL
LIN {X 0,Y 512.192,Z 555.556,A -85,B 0,C 180,E1 -5415.401,E2 -5415.401} C_VEL
LIN {X 0,Y 510.608,Z 545.338,A -85,B 0,C 180,E1 -5415.624,E2 -5415.624} C_VEL
LIN {X 0,Y 510.991,Z 526.858,A -85,B 0,C 180,E1 -5418.239,E2 -5418.239} C_VEL
LIN {X 0,Y 511.445,Z 506.137,A -85,B 0,C 180,E1 -5421.144,E2 -5421.144} C_VEL
LIN {X 0,Y 511.832,Z 482.941,A -85,B 0,C 180,E1 -5424.326,E2 -5424.326} C_VEL
LIN {X 0,Y 509.905,Z 472.096,A -85,B 0,C 180,E1 -5425.897,E2 -5425.897} C_VEL
LIN {X 0,Y 509.879,Z 472.101,A -85,B 0,C 180,E1 -5428.844,E2 -5428.844} C_VEL
LIN {X 0,Y 509.823,Z 472.104,A -85,B 0,C 180,E1 -5431.59,E2 -5431.59} C_VEL
LIN {X 0,Y 509.85,Z 472.104,A -85,B 0,C 180,E1 -5434.414,E2 -5434.414} C_VEL
LIN {X 0,Y 509.819,Z 472.103,A -85,B 0,C 180,E1 -5437.341,E2 -5437.341} C_VEL
LIN {X 0,Y 509.84,Z 472.104,A -85,B 0,C 180,E1 -5440.382,E2 -5440.382} C_VEL
LIN {X 0,Y 509.824,Z 472.102,A -85,B 0,C 180,E1 -5443.062,E2 -5443.062} C_VEL
LIN {X 0,Y 509.833,Z 472.099,A -85,B 0,C 180,E1 -5445.792,E2 -5445.792} C_VEL
LIN {X 0,Y 509.86,Z 472.102,A -85,B 0,C 180,E1 -5448.575,E2 -5448.575} C_VEL
LIN {X 0,Y 509.853,Z 472.098,A -85,B 0,C 180,E1 -5451.786,E2 -5451.786} C_VEL
LIN {X 0,Y 509.847,Z 472.104,A -85,B 0,C 180,E1 -5454.623,E2 -5454.623} C_VEL
LIN {X 0,Y 509.868,Z 472.095,A -85,B 0,C 180,E1 -5457.481,E2 -5457.481} C_VEL
LIN {X 0,Y 509.884,Z 472.1,A -85,B 0,C 180,E1 -5460.269,E2 -5460.269} C_VEL
LIN {X 0,Y 509.887,Z 472.097,A -85,B 0,C 180,E1 -5462.944,E2 -5462.944} C_VEL
LIN {X 0,Y 509.943,Z 472.285,A -85,B 0,C 180,E1 -5464.16,E2 -5464.16} C_VEL
LIN {X 0,Y 512.874,Z 485.771,A -85,B 0,C 180,E1 -5466.156,E2 -5466.156} C_VEL
LIN {X 0,Y 511.973,Z 509.686,A -85,B 0,C 180,E1 -5469.3,E2 -5469.3} C_VEL
LIN {X 0,Y 511.494,Z 524.325,A -85,B 0,C 180,E1 -5471.211,E2 -5471.211} C_VEL
LIN {X 0,Y 513.506,Z 536.665,A -85,B 0,C 180,E1 -5471.477,E2 -5471.477} C_VEL
LIN {X 0,Y 512.667,Z 656.023,A -85,B 0,C 180,E1 -5473.192,E2 -5473.192} C_VEL
LIN {X 0,Y 512.442,Z 670.856,A -85,B 0,C 180,E1 -5473.499,E2 -5473.499} C_VEL
LIN {X 0,Y 512.149,Z 685.273,A -85,B 0,C 180,E1 -5473.968,E2 -5473.968} C_VEL
LIN {X 0,Y 511.777,Z 698.699,A -85,B 0,C 180,E1 -5474.57,E2 -5474.57} C_VEL
LIN {X 0,Y 511.401,Z 710.888,A -85,B 0,C 180,E1 -5475.271,E2 -5475.271} C_VEL
LIN {X 0,Y 510.947,Z 723.489,A -85,B 0,C 180,E1 -5476.173,E2 -5476.173} C_VEL
LIN {X 0,Y 510.541,Z 734.864,A -85,B 0,C 180,E1 -5477.175,E2 -5477.175} C_VEL
LIN {X 0,Y 510.214,Z 745.166,A -85,B 0,C 180,E1 -5478.277,E2 -5478.277} C_VEL
LIN {X 0,Y 509.901,Z 754.471,A -85,B 0,C 180,E1 -5479.477,E2 -5479.477} C_VEL
LIN {X 0,Y 509.601,Z 763.34,A -85,B 0,C 180,E1 -5480.874,E2 -5480.874} C_VEL
LIN {X 0,Y 509.424,Z 769.586,A -85,B 0,C 180,E1 -5482.07,E2 -5482.07} C_VEL
LIN {X 0,Y 509.308,Z 776.201,A -85,B 0,C 180,E1 -5483.662,E2 -5483.662} C_VEL
LIN {X 0,Y 509.239,Z 780.073,A -85,B 0,C 180,E1 -5484.853,E2 -5484.853} C_VEL
LIN {X 0,Y 509.218,Z 783.045,A -85,B 0,C 180,E1 -5486.043,E2 -5486.043} C_VEL
LIN {X 0,Y 509.187,Z 785.769,A -85,B 0,C 180,E1 -5487.627,E2 -5487.627} C_VEL
LIN {X 0,Y 509.071,Z 787.115,A -85,B 0,C 180,E1 -5489.209,E2 -5489.209} C_VEL
LIN {X 0,Y 509.071,Z 787.113,A -85,B 0,C 180,E1 -5490.791,E2 -5490.791} C_VEL
LIN {X 0,Y 509.187,Z 785.764,A -85,B 0,C 180,E1 -5492.373,E2 -5492.373} C_VEL
LIN {X 0,Y 509.218,Z 783.035,A -85,B 0,C 180,E1 -5493.957,E2 -5493.957} C_VEL
LIN {X 0,Y 509.301,Z 778.848,A -85,B 0,C 180,E1 -5495.543,E2 -5495.543} C_VEL
LIN {X 0,Y 509.328,Z 773.069,A -85,B 0,C 180,E1 -5497.134,E2 -5497.134} C_VEL
LIN {X 0,Y 509.519,Z 766.543,A -85,B 0,C 180,E1 -5498.527,E2 -5498.527} C_VEL
LIN {X 0,Y 509.753,Z 758.411,A -85,B 0,C 180,E1 -5499.924,E2 -5499.924} C_VEL
LIN {X 0,Y 510.02,Z 749.88,A -85,B 0,C 180,E1 -5501.123,E2 -5501.123} C_VEL
LIN {X 0,Y 510.365,Z 739.943,A -85,B 0,C 180,E1 -5502.284,E2 -5502.284} C_VEL
LIN {X 0,Y 510.731,Z 729.147,A -85,B 0,C 180,E1 -5503.326,E2 -5503.326} C_VEL
LIN {X 0,Y 511.099,Z 717.813,A -85,B 0,C 180,E1 -5504.229,E2 -5504.229} C_VEL
LIN {X 0,Y 511.548,Z 705.425,A -85,B 0,C 180,E1 -5505.03,E2 -5505.03} C_VEL
LIN {X 0,Y 511.884,Z 692.736,A -85,B 0,C 180,E1 -5505.682,E2 -5505.682} C_VEL
LIN {X 0,Y 512.218,Z 678.518,A -85,B 0,C 180,E1 -5506.234,E2 -5506.234} C_VEL
LIN {X 0,Y 512.493,Z 664.38,A -85,B 0,C 180,E1 -5506.614,E2 -5506.614} C_VEL
LIN {X 0,Y 512.681,Z 638.867,A -85,B 0,C 180,E1 -5507.013,E2 -5507.013} C_VEL
LIN {X 0,Y 513.324,Z 536.143,A -85,B 0,C 180,E1 -5508.501,E2 -5508.501} C_VEL
LIN {X 0,Y 511.482,Z 524.514,A -85,B 0,C 180,E1 -5508.751,E2 -5508.751} C_VEL
LIN {X 0,Y 512.372,Z 498.505,A -85,B 0,C 180,E1 -5512.161,E2 -5512.161} C_VEL
LIN {X 0,Y 512.948,Z 486.027,A -85,B 0,C 180,E1 -5513.84,E2 -5513.84} C_VEL
LIN {X 0,Y 511.078,Z 476.863,A -85,B 0,C 180,E1 -5515.233,E2 -5515.233} C_VEL
LIN {X 0,Y 509.906,Z 472.097,A -85,B 0,C 180,E1 -5516.006,E2 -5516.006} C_VEL
LIN {X 0,Y 509.88,Z 472.099,A -85,B 0,C 180,E1 -5518.844,E2 -5518.844} C_VEL
LIN {X 0,Y 509.827,Z 472.108,A -85,B 0,C 180,E1 -5521.59,E2 -5521.59} C_VEL
LIN {X 0,Y 509.85,Z 472.099,A -85,B 0,C 180,E1 -5524.414,E2 -5524.414} C_VEL
LIN {X 0,Y 509.819,Z 472.109,A -85,B 0,C 180,E1 -5527.341,E2 -5527.341} C_VEL
LIN {X 0,Y 509.841,Z 472.1,A -85,B 0,C 180,E1 -5530.382,E2 -5530.382} C_VEL
LIN {X 0,Y 509.843,Z 472.105,A -85,B 0,C 180,E1 -5533.064,E2 -5533.064} C_VEL
LIN {X 0,Y 509.833,Z 472.101,A -85,B 0,C 180,E1 -5535.793,E2 -5535.793} C_VEL
LIN {X 0,Y 509.86,Z 472.1,A -85,B 0,C 180,E1 -5538.575,E2 -5538.575} C_VEL
LIN {X 0,Y 509.855,Z 472.099,A -85,B 0,C 180,E1 -5541.786,E2 -5541.786} C_VEL
LIN {X 0,Y 509.837,Z 472.105,A -85,B 0,C 180,E1 -5544.622,E2 -5544.622} C_VEL
LIN {X 0,Y 509.867,Z 472.098,A -85,B 0,C 180,E1 -5547.481,E2 -5547.481} C_VEL
LIN {X 0,Y 509.862,Z 472.102,A -85,B 0,C 180,E1 -5550.274,E2 -5550.274} C_VEL
LIN {X 0,Y 509.889,Z 472.105,A -85,B 0,C 180,E1 -5552.945,E2 -5552.945} C_VEL
LIN {X 0,Y 509.882,Z 472.183,A -85,B 0,C 180,E1 -5554.622,E2 -5554.622} C_VEL
LIN {X 0,Y 512.3,Z 483.305,A -85,B 0,C 180,E1 -5556.557,E2 -5556.557} C_VEL
LIN {X 0,Y 511.983,Z 495.511,A -85,B 0,C 180,E1 -5558.457,E2 -5558.457} C_VEL
LIN {X 0,Y 511.269,Z 515.941,A -85,B 0,C 180,E1 -5561.569,E2 -5561.569} C_VEL
LIN {X 0,Y 510.642,Z 539.155,A -85,B 0,C 180,E1 -5565.045,E2 -5565.045} C_VEL
LIN {X 0,Y 510.572,Z 541.207,A -85,B 0,C 180,E1 -5565.349,E2 -5565.349} C_VEL
LIN {X 0,Y 512.394,Z 552.819,A -85,B 0,C 180,E1 -5565.605,E2 -5565.605} C_VEL
LIN {X 0,Y 511.649,Z 651.927,A -85,B 0,C 180,E1 -5567.123,E2 -5567.123} C_VEL
LIN {X 0,Y 511.452,Z 665.224,A -85,B 0,C 180,E1 -5567.489,E2 -5567.489} C_VEL
LIN {X 0,Y 511.2,Z 678.207,A -85,B 0,C 180,E1 -5568.018,E2 -5568.018} C_VEL
LIN {X 0,Y 510.937,Z 690.455,A -85,B 0,C 180,E1 -5568.696,E2 -5568.696} C_VEL
LIN {X 0,Y 510.507,Z 701.695,A -85,B 0,C 180,E1 -5569.49,E2 -5569.49} C_VEL
LIN {X 0,Y 510.206,Z 711.808,A -85,B 0,C 180,E1 -5570.385,E2 -5570.385} C_VEL
LIN {X 0,Y 509.912,Z 721.755,A -85,B 0,C 180,E1 -5571.479,E2 -5571.479} C_VEL
LIN {X 0,Y 509.65,Z 730.483,A -85,B 0,C 180,E1 -5572.672,E2 -5572.672} C_VEL
LIN {X 0,Y 509.561,Z 737.471,A -85,B 0,C 180,E1 -5573.864,E2 -5573.864} C_VEL
LIN {X 0,Y 509.278,Z 743.853,A -85,B 0,C 180,E1 -5575.25,E2 -5575.25} C_VEL
LIN {X 0,Y 509.276,Z 748.029,A -85,B 0,C 180,E1 -5576.44,E2 -5576.44} C_VEL
LIN {X 0,Y 509.21,Z 751.168,A -85,B 0,C 180,E1 -5577.627,E2 -5577.627} C_VEL
LIN {X 0,Y 509.118,Z 752.712,A -85,B 0,C 180,E1 -5578.418,E2 -5578.418} C_VEL
LIN {X 0,Y 509.075,Z 753.841,A -85,B 0,C 180,E1 -5579.209,E2 -5579.209} C_VEL
LIN {X 0,Y 509.066,Z 754.558,A -85,B 0,C 180,E1 -5580,E2 -5580} C_VEL
LIN {X 0,Y 509.112,Z 754.788,A -85,B 0,C 180,E1 -5581.582,E2 -5581.582} C_VEL
LIN {X 0,Y 509.188,Z 754.316,A -85,B 0,C 180,E1 -5582.373,E2 -5582.373} C_VEL
LIN {X 0,Y 509.193,Z 753.441,A -85,B 0,C 180,E1 -5583.165,E2 -5583.165} C_VEL
LIN {X 0,Y 509.257,Z 752.149,A -85,B 0,C 180,E1 -5583.957,E2 -5583.957} C_VEL
LIN {X 0,Y 509.228,Z 749.457,A -85,B 0,C 180,E1 -5585.147,E2 -5585.147} C_VEL
LIN {X 0,Y 509.27,Z 745.194,A -85,B 0,C 180,E1 -5586.477,E2 -5586.477} C_VEL
LIN {X 0,Y 509.378,Z 740.836,A -85,B 0,C 180,E1 -5587.532,E2 -5587.532} C_VEL
LIN {X 0,Y 509.54,Z 734.665,A -85,B 0,C 180,E1 -5588.727,E2 -5588.727} C_VEL
LIN {X 0,Y 509.705,Z 726.967,A -85,B 0,C 180,E1 -5589.925,E2 -5589.925} C_VEL
LIN {X 0,Y 510.025,Z 719.123,A -85,B 0,C 180,E1 -5590.922,E2 -5590.922} C_VEL
LIN {X 0,Y 510.197,Z 709.51,A -85,B 0,C 180,E1 -5591.925,E2 -5591.925} C_VEL
LIN {X 0,Y 510.598,Z 698.779,A -85,B 0,C 180,E1 -5592.823,E2 -5592.823} C_VEL
LIN {X 0,Y 510.991,Z 686.739,A -85,B 0,C 180,E1 -5593.623,E2 -5593.623} C_VEL
LIN {X 0,Y 511.287,Z 673.905,A -85,B 0,C 180,E1 -5594.274,E2 -5594.274} C_VEL
LIN {X 0,Y 511.5,Z 660.833,A -85,B 0,C 180,E1 -5594.751,E2 -5594.751} C_VEL
LIN {X 0,Y 511.721,Z 647.919,A -85,B 0,C 180,E1 -5595.05,E2 -5595.05} C_VEL
LIN {X 0,Y 512.31,Z 552.816,A -85,B 0,C 180,E1 -5596.453,E2 -5596.453} C_VEL
LIN {X 0,Y 510.539,Z 541.412,A -85,B 0,C 180,E1 -5596.702,E2 -5596.702} C_VEL
LIN {X 0,Y 511.059,Z 522.805,A -85,B 0,C 180,E1 -5599.48,E2 -5599.48} C_VEL
LIN {X 0,Y 511.657,Z 503.465,A -85,B 0,C 180,E1 -5602.406,E2 -5602.406} C_VEL
LIN {X 0,Y 512.297,Z 485.462,A -85,B 0,C 180,E1 -5605.168,E2 -5605.168} C_VEL
LIN {X 0,Y 511.913,Z 481.298,A -85,B 0,C 180,E1 -5605.842,E2 -5605.842} C_VEL
LIN {X 0,Y 509.892,Z 472.099,A -85,B 0,C 180,E1 -5607.444,E2 -5607.444} C_VEL
LIN {X 0,Y 509.861,Z 472.103,A -85,B 0,C 180,E1 -5609.751,E2 -5609.751} C_VEL
LIN {X 0,Y 509.876,Z 472.095,A -85,B 0,C 180,E1 -5612.774,E2 -5612.774} C_VEL
LIN {X 0,Y 509.832,Z 472.099,A -85,B 0,C 180,E1 -5614.777,E2 -5614.777} C_VEL
LIN {X 0,Y 509.156,Z 472.189,A -85,B 0,C 180,E1 -5615.437,E2 -5615.437} C_VEL
LIN {X 0,Y 506.299,Z 472.544,A -85,B 0,C 180,E1 -5616.508,E2 -5616.508} C_VEL
LIN {X 0,Y 503.894,Z 472.843,A -85,B 0,C 180,E1 -5617.371,E2 -5617.371} C_VEL
LIN {X 0,Y 502.871,Z 472.969,A -85,B 0,C 180,E1 -5618.037,E2 -5618.037} C_VEL
LIN {X 0,Y 502.792,Z 472.976,A -85,B 0,C 180,E1 -5618.263,E2 -5618.263} C_VEL
LIN {X 0,Y 502.822,Z 472.973,A -85,B 0,C 180,E1 -5621.066,E2 -5621.066} C_VEL
LIN {X 0,Y 502.788,Z 472.975,A -85,B 0,C 180,E1 -5624.53,E2 -5624.53} C_VEL
LIN {X 0,Y 502.799,Z 472.979,A -85,B 0,C 180,E1 -5627.861,E2 -5627.861} C_VEL
LIN {X 0,Y 502.803,Z 472.975,A -85,B 0,C 180,E1 -5631.024,E2 -5631.024} C_VEL
LIN {X 0,Y 502.777,Z 472.978,A -85,B 0,C 180,E1 -5634.169,E2 -5634.169} C_VEL
LIN {X 0,Y 502.834,Z 472.971,A -85,B 0,C 180,E1 -5636.993,E2 -5636.993} C_VEL
LIN {X 0,Y 502.817,Z 472.974,A -85,B 0,C 180,E1 -5640.065,E2 -5640.065} C_VEL
LIN {X 0,Y 502.835,Z 472.969,A -85,B 0,C 180,E1 -5642.533,E2 -5642.533} C_VEL
LIN {X 0,Y 502.829,Z 472.976,A -85,B 0,C 180,E1 -5645.299,E2 -5645.299} C_VEL
LIN {X 0,Y 502.782,Z 472.98,A -85,B 0,C 180,E1 -5647.826,E2 -5647.826} C_VEL
LIN {X 0,Y 502.827,Z 472.97,A -85,B 0,C 180,E1 -5650.4,E2 -5650.4} C_VEL
LIN {X 0,Y 502.837,Z 472.971,A -85,B 0,C 180,E1 -5652.932,E2 -5652.932} C_VEL
LIN {X 0,Y 502.854,Z 472.975,A -85,B 0,C 180,E1 -5655.429,E2 -5655.429} C_VEL
LIN {X 0,Y 502.88,Z 472.964,A -85,B 0,C 180,E1 -5658.717,E2 -5658.717} C_VEL
LIN {X 0,Y 502.905,Z 472.963,A -85,B 0,C 180,E1 -5661.967,E2 -5661.967} C_VEL
LIN {X 0,Y 502.94,Z 472.956,A -85,B 0,C 180,E1 -5664.386,E2 -5664.386} C_VEL
LIN {X 0,Y 503.028,Z 472.952,A -85,B 0,C 180,E1 -5667.598,E2 -5667.598} C_VEL
LIN {X 0,Y 503.03,Z 472.947,A -85,B 0,C 180,E1 -5670,E2 -5670} C_VEL
LIN {X 0,Y 503.028,Z 472.945,A -85,B 0,C 180,E1 -5672.402,E2 -5672.402} C_VEL
LIN {X 0,Y 502.936,Z 472.963,A -85,B 0,C 180,E1 -5675.613,E2 -5675.613} C_VEL
LIN {X 0,Y 502.904,Z 472.962,A -85,B 0,C 180,E1 -5678.033,E2 -5678.033} C_VEL
LIN {X 0,Y 502.879,Z 472.971,A -85,B 0,C 180,E1 -5681.283,E2 -5681.283} C_VEL
LIN {X 0,Y 502.847,Z 472.968,A -85,B 0,C 180,E1 -5684.571,E2 -5684.571} C_VEL
LIN {X 0,Y 502.864,Z 472.968,A -85,B 0,C 180,E1 -5687.907,E2 -5687.907} C_VEL
LIN {X 0,Y 502.83,Z 472.97,A -85,B 0,C 180,E1 -5690.536,E2 -5690.536} C_VEL
LIN {X 0,Y 502.799,Z 472.978,A -85,B 0,C 180,E1 -5693.04,E2 -5693.04} C_VEL
LIN {X 0,Y 502.843,Z 472.973,A -85,B 0,C 180,E1 -5695.676,E2 -5695.676} C_VEL
LIN {X 0,Y 502.842,Z 472.968,A -85,B 0,C 180,E1 -5698.373,E2 -5698.373} C_VEL
LIN {X 0,Y 502.795,Z 472.981,A -85,B 0,C 180,E1 -5701.499,E2 -5701.499} C_VEL
LIN {X 0,Y 502.805,Z 472.974,A -85,B 0,C 180,E1 -5703.994,E2 -5703.994} C_VEL
LIN {X 0,Y 502.779,Z 472.983,A -85,B 0,C 180,E1 -5707.178,E2 -5707.178} C_VEL
LIN {X 0,Y 502.79,Z 472.976,A -85,B 0,C 180,E1 -5710.015,E2 -5710.015} C_VEL
LIN {X 0,Y 502.805,Z 472.973,A -85,B 0,C 180,E1 -5712.199,E2 -5712.199} C_VEL
LIN {X 0,Y 502.803,Z 472.98,A -85,B 0,C 180,E1 -5715.468,E2 -5715.468} C_VEL
LIN {X 0,Y 502.821,Z 472.975,A -85,B 0,C 180,E1 -5718.934,E2 -5718.934} C_VEL
LIN {X 0,Y 502.796,Z 472.975,A -85,B 0,C 180,E1 -5722.046,E2 -5722.046} C_VEL
LIN {X 0,Y 502.803,Z 472.979,A -85,B 0,C 180,E1 -5725.035,E2 -5725.035} C_VEL
LIN {X 0,Y 502.786,Z 472.978,A -85,B 0,C 180,E1 -5727.916,E2 -5727.916} C_VEL
LIN {X 0,Y 502.827,Z 472.973,A -85,B 0,C 180,E1 -5730.712,E2 -5730.712} C_VEL
LIN {X 0,Y 502.886,Z 472.991,A -85,B 0,C 180,E1 -5733.625,E2 -5733.625} C_VEL
LIN {X 0,Y 505.236,Z 485.376,A -85,B 0,C 180,E1 -5735.554,E2 -5735.554} C_VEL
LIN {X 0,Y 504.643,Z 506.066,A -85,B 0,C 180,E1 -5738.557,E2 -5738.557} C_VEL
LIN {X 0,Y 504.122,Z 526.854,A -85,B 0,C 180,E1 -5741.579,E2 -5741.579} C_VEL
LIN {X 0,Y 503.671,Z 545.36,A -85,B 0,C 180,E1 -5744.256,E2 -5744.256} C_VEL
LIN {X 0,Y 505.366,Z 556.955,A -85,B 0,C 180,E1 -5744.496,E2 -5744.496} C_VEL
LIN {X 0,Y 504.726,Z 655.014,A -85,B 0,C 180,E1 -5745.973,E2 -5745.973} C_VEL
LIN {X 0,Y 504.54,Z 667.267,A -85,B 0,C 180,E1 -5746.302,E2 -5746.302} C_VEL
LIN {X 0,Y 504.225,Z 679.946,A -85,B 0,C 180,E1 -5746.807,E2 -5746.807} C_VEL
LIN {X 0,Y 503.888,Z 692.878,A -85,B 0,C 180,E1 -5747.51,E2 -5747.51} C_VEL
LIN {X 0,Y 503.554,Z 704.326,A -85,B 0,C 180,E1 -5748.324,E2 -5748.324} C_VEL
LIN {X 0,Y 503.18,Z 715.592,A -85,B 0,C 180,E1 -5749.335,E2 -5749.335} C_VEL
LIN {X 0,Y 502.902,Z 724.639,A -85,B 0,C 180,E1 -5750.346,E2 -5750.346} C_VEL
LIN {X 0,Y 502.594,Z 733.413,A -85,B 0,C 180,E1 -5751.557,E2 -5751.557} C_VEL
LIN {X 0,Y 502.408,Z 740.476,A -85,B 0,C 180,E1 -5752.767,E2 -5752.767} C_VEL
LIN {X 0,Y 502.338,Z 746.09,A -85,B 0,C 180,E1 -5753.977,E2 -5753.977} C_VEL
LIN {X 0,Y 502.117,Z 750.489,A -85,B 0,C 180,E1 -5755.183,E2 -5755.183} C_VEL
LIN {X 0,Y 502.218,Z 752.797,A -85,B 0,C 180,E1 -5755.988,E2 -5755.988} C_VEL
LIN {X 0,Y 502.124,Z 754.685,A -85,B 0,C 180,E1 -5756.791,E2 -5756.791} C_VEL
LIN {X 0,Y 502.12,Z 756.139,A -85,B 0,C 180,E1 -5757.593,E2 -5757.593} C_VEL
LIN {X 0,Y 501.991,Z 757.784,A -85,B 0,C 180,E1 -5759.198,E2 -5759.198} C_VEL
LIN {X 0,Y 501.98,Z 758.031,A -85,B 0,C 180,E1 -5760,E2 -5760} C_VEL
LIN {X 0,Y 501.991,Z 757.845,A -85,B 0,C 180,E1 -5760.802,E2 -5760.802} C_VEL
LIN {X 0,Y 502.12,Z 756.286,A -85,B 0,C 180,E1 -5762.407,E2 -5762.407} C_VEL
LIN {X 0,Y 502.125,Z 754.908,A -85,B 0,C 180,E1 -5763.209,E2 -5763.209} C_VEL
LIN {X 0,Y 502.187,Z 752.012,A -85,B 0,C 180,E1 -5764.415,E2 -5764.415} C_VEL
LIN {X 0,Y 502.283,Z 748.068,A -85,B 0,C 180,E1 -5765.621,E2 -5765.621} C_VEL
LIN {X 0,Y 502.365,Z 742.064,A -85,B 0,C 180,E1 -5767.011,E2 -5767.011} C_VEL
LIN {X 0,Y 502.555,Z 735.294,A -85,B 0,C 180,E1 -5768.241,E2 -5768.241} C_VEL
LIN {X 0,Y 502.799,Z 726.949,A -85,B 0,C 180,E1 -5769.453,E2 -5769.453} C_VEL
LIN {X 0,Y 503.051,Z 718.363,A -85,B 0,C 180,E1 -5770.464,E2 -5770.464} C_VEL
LIN {X 0,Y 503.425,Z 707.809,A -85,B 0,C 180,E1 -5771.475,E2 -5771.475} C_VEL
LIN {X 0,Y 503.768,Z 696.783,A -85,B 0,C 180,E1 -5772.313,E2 -5772.313} C_VEL
LIN {X 0,Y 504.038,Z 685.472,A -85,B 0,C 180,E1 -5772.993,E2 -5772.993} C_VEL
LIN {X 0,Y 504.314,Z 673.386,A -85,B 0,C 180,E1 -5773.55,E2 -5773.55} C_VEL
LIN {X 0,Y 504.59,Z 659.937,A -85,B 0,C 180,E1 -5773.979,E2 -5773.979} C_VEL
LIN {X 0,Y 504.774,Z 647.033,A -85,B 0,C 180,E1 -5774.231,E2 -5774.231} C_VEL
LIN {X 0,Y 505.299,Z 555.975,A -85,B 0,C 180,E1 -5775.605,E2 -5775.605} C_VEL
LIN {X 0,Y 503.666,Z 545.655,A -85,B 0,C 180,E1 -5775.831,E2 -5775.831} C_VEL
LIN {X 0,Y 504.103,Z 525.414,A -85,B 0,C 180,E1 -5778.703,E2 -5778.703} C_VEL
LIN {X 0,Y 504.49,Z 507.332,A -85,B 0,C 180,E1 -5781.236,E2 -5781.236} C_VEL
LIN {X 0,Y 504.914,Z 485.638,A -85,B 0,C 180,E1 -5784.244,E2 -5784.244} C_VEL
LIN {X 0,Y 504.269,Z 479.937,A -85,B 0,C 180,E1 -5785.054,E2 -5785.054} C_VEL
LIN {X 0,Y 502.875,Z 472.973,A -85,B 0,C 180,E1 -5786.091,E2 -5786.091} C_VEL
LIN {X 0,Y 502.827,Z 472.977,A -85,B 0,C 180,E1 -5789.288,E2 -5789.288} C_VEL
LIN {X 0,Y 502.786,Z 472.982,A -85,B 0,C 180,E1 -5792.084,E2 -5792.084} C_VEL
LIN {X 0,Y 502.802,Z 472.981,A -85,B 0,C 180,E1 -5794.966,E2 -5794.966} C_VEL
LIN {X 0,Y 502.796,Z 472.978,A -85,B 0,C 180,E1 -5797.954,E2 -5797.954} C_VEL
LIN {X 0,Y 502.822,Z 472.975,A -85,B 0,C 180,E1 -5801.066,E2 -5801.066} C_VEL
LIN {X 0,Y 502.803,Z 472.982,A -85,B 0,C 180,E1 -5804.532,E2 -5804.532} C_VEL
LIN {X 0,Y 502.832,Z 472.972,A -85,B 0,C 180,E1 -5807.864,E2 -5807.864} C_VEL
LIN {X 0,Y 502.803,Z 472.977,A -85,B 0,C 180,E1 -5811.024,E2 -5811.024} C_VEL
LIN {X 0,Y 502.787,Z 472.983,A -85,B 0,C 180,E1 -5814.167,E2 -5814.167} C_VEL
LIN {X 0,Y 502.835,Z 472.973,A -85,B 0,C 180,E1 -5816.993,E2 -5816.993} C_VEL
LIN {X 0,Y 502.833,Z 472.977,A -85,B 0,C 180,E1 -5820.062,E2 -5820.062} C_VEL
LIN {X 0,Y 502.836,Z 472.978,A -85,B 0,C 180,E1 -5822.533,E2 -5822.533} C_VEL
LIN {X 0,Y 502.898,Z 473.112,A -85,B 0,C 180,E1 -5823.882,E2 -5823.882} C_VEL
LIN {X 0,Y 506.036,Z 487.353,A -85,B 0,C 180,E1 -5826.031,E2 -5826.031} C_VEL
LIN {X 0,Y 505.056,Z 511.272,A -85,B 0,C 180,E1 -5829.223,E2 -5829.223} C_VEL
LIN {X 0,Y 504.603,Z 524.491,A -85,B 0,C 180,E1 -5830.966,E2 -5830.966} C_VEL
LIN {X 0,Y 506.686,Z 538.13,A -85,B 0,C 180,E1 -5831.258,E2 -5831.258} C_VEL
LIN {X 0,Y 505.804,Z 657.035,A -85,B 0,C 180,E1 -5833.009,E2 -5833.009} C_VEL
LIN {X 0,Y 505.523,Z 672.158,A -85,B 0,C 180,E1 -5833.34,E2 -5833.34} C_VEL
LIN {X 0,Y 505.249,Z 685.618,A -85,B 0,C 180,E1 -5833.795,E2 -5833.795} C_VEL
LIN {X 0,Y 504.885,Z 697.929,A -85,B 0,C 180,E1 -5834.354,E2 -5834.354} C_VEL
LIN {X 0,Y 504.499,Z 710.246,A -85,B 0,C 180,E1 -5835.065,E2 -5835.065} C_VEL
LIN {X 0,Y 504.067,Z 721.635,A -85,B 0,C 180,E1 -5835.878,E2 -5835.878} C_VEL
LIN {X 0,Y 503.586,Z 733.315,A -85,B 0,C 180,E1 -5836.892,E2 -5836.892} C_VEL
LIN {X 0,Y 503.255,Z 742.98,A -85,B 0,C 180,E1 -5837.908,E2 -5837.908} C_VEL
LIN {X 0,Y 502.909,Z 752.659,A -85,B 0,C 180,E1 -5839.125,E2 -5839.125} C_VEL
LIN {X 0,Y 502.61,Z 761.889,A -85,B 0,C 180,E1 -5840.543,E2 -5840.543} C_VEL
LIN {X 0,Y 502.364,Z 769.291,A -85,B 0,C 180,E1 -5841.958,E2 -5841.958} C_VEL
LIN {X 0,Y 502.234,Z 775.931,A -85,B 0,C 180,E1 -5843.572,E2 -5843.572} C_VEL
LIN {X 0,Y 502.172,Z 779.823,A -85,B 0,C 180,E1 -5844.781,E2 -5844.781} C_VEL
LIN {X 0,Y 502.113,Z 782.803,A -85,B 0,C 180,E1 -5845.987,E2 -5845.987} C_VEL
LIN {X 0,Y 502.089,Z 785.54,A -85,B 0,C 180,E1 -5847.593,E2 -5847.593} C_VEL
LIN {X 0,Y 501.988,Z 786.891,A -85,B 0,C 180,E1 -5849.198,E2 -5849.198} C_VEL
LIN {X 0,Y 501.988,Z 786.886,A -85,B 0,C 180,E1 -5850.802,E2 -5850.802} C_VEL
LIN {X 0,Y 502.089,Z 785.526,A -85,B 0,C 180,E1 -5852.407,E2 -5852.407} C_VEL
LIN {X 0,Y 502.113,Z 782.778,A -85,B 0,C 180,E1 -5854.013,E2 -5854.013} C_VEL
LIN {X 0,Y 502.213,Z 778.567,A -85,B 0,C 180,E1 -5855.622,E2 -5855.622} C_VEL
LIN {X 0,Y 502.254,Z 772.756,A -85,B 0,C 180,E1 -5857.235,E2 -5857.235} C_VEL
LIN {X 0,Y 502.438,Z 766.187,A -85,B 0,C 180,E1 -5858.648,E2 -5858.648} C_VEL
LIN {X 0,Y 502.705,Z 758.006,A -85,B 0,C 180,E1 -5860.064,E2 -5860.064} C_VEL
LIN {X 0,Y 502.978,Z 749.42,A -85,B 0,C 180,E1 -5861.281,E2 -5861.281} C_VEL
LIN {X 0,Y 503.356,Z 739.406,A -85,B 0,C 180,E1 -5862.458,E2 -5862.458} C_VEL
LIN {X 0,Y 503.729,Z 728.503,A -85,B 0,C 180,E1 -5863.515,E2 -5863.515} C_VEL
LIN {X 0,Y 504.124,Z 717.053,A -85,B 0,C 180,E1 -5864.43,E2 -5864.43} C_VEL
LIN {X 0,Y 504.628,Z 704.514,A -85,B 0,C 180,E1 -5865.241,E2 -5865.241} C_VEL
LIN {X 0,Y 505.008,Z 690.454,A -85,B 0,C 180,E1 -5865.953,E2 -5865.953} C_VEL
LIN {X 0,Y 505.342,Z 676.573,A -85,B 0,C 180,E1 -5866.477,E2 -5866.477} C_VEL
LIN {X 0,Y 505.64,Z 661.762,A -85,B 0,C 180,E1 -5866.856,E2 -5866.856} C_VEL
LIN {X 0,Y 506.546,Z 537.141,A -85,B 0,C 180,E1 -5868.716,E2 -5868.716} C_VEL
LIN {X 0,Y 504.593,Z 524.573,A -85,B 0,C 180,E1 -5869.002,E2 -5869.002} C_VEL
LIN {X 0,Y 505.511,Z 500.158,A -85,B 0,C 180,E1 -5872.263,E2 -5872.263} C_VEL
LIN {X 0,Y 506.148,Z 487.779,A -85,B 0,C 180,E1 -5873.963,E2 -5873.963} C_VEL
LIN {X 0,Y 503.927,Z 477.221,A -85,B 0,C 180,E1 -5875.616,E2 -5875.616} C_VEL
LIN {X 0,Y 502.869,Z 472.973,A -85,B 0,C 180,E1 -5876.34,E2 -5876.34} C_VEL
LIN {X 0,Y 502.827,Z 472.98,A -85,B 0,C 180,E1 -5879.288,E2 -5879.288} C_VEL
LIN {X 0,Y 502.789,Z 472.981,A -85,B 0,C 180,E1 -5882.084,E2 -5882.084} C_VEL
LIN {X 0,Y 502.801,Z 472.98,A -85,B 0,C 180,E1 -5884.966,E2 -5884.966} C_VEL
LIN {X 0,Y 502.795,Z 472.979,A -85,B 0,C 180,E1 -5887.954,E2 -5887.954} C_VEL
LIN {X 0,Y 502.822,Z 472.979,A -85,B 0,C 180,E1 -5891.066,E2 -5891.066} C_VEL
LIN {X 0,Y 502.785,Z 472.983,A -85,B 0,C 180,E1 -5893.376,E2 -5893.376} C_VEL
LIN {X 0,Y 502.793,Z 472.979,A -85,B 0,C 180,E1 -5895.661,E2 -5895.661} C_VEL
LIN {X 0,Y 502.822,Z 472.979,A -85,B 0,C 180,E1 -5899.005,E2 -5899.005} C_VEL
LIN {X 0,Y 502.797,Z 472.978,A -85,B 0,C 180,E1 -5902.046,E2 -5902.046} C_VEL
LIN {X 0,Y 502.806,Z 472.981,A -85,B 0,C 180,E1 -5905.035,E2 -5905.035} C_VEL
LIN {X 0,Y 502.789,Z 472.979,A -85,B 0,C 180,E1 -5907.916,E2 -5907.916} C_VEL
LIN {X 0,Y 502.828,Z 472.982,A -85,B 0,C 180,E1 -5910.712,E2 -5910.712} C_VEL
LIN {X 0,Y 502.866,Z 472.978,A -85,B 0,C 180,E1 -5913.881,E2 -5913.881} C_VEL
LIN {X 0,Y 502.874,Z 473.096,A -85,B 0,C 180,E1 -5914.326,E2 -5914.326} C_VEL
LIN {X 0,Y 505.495,Z 485.179,A -85,B 0,C 180,E1 -5916.476,E2 -5916.476} C_VEL
LIN {X 0,Y 505.041,Z 498.45,A -85,B 0,C 180,E1 -5918.575,E2 -5918.575} C_VEL
LIN {X 0,Y 504.32,Z 517.433,A -85,B 0,C 180,E1 -5921.511,E2 -5921.511} C_VEL
LIN {X 0,Y 503.696,Z 539.303,A -85,B 0,C 180,E1 -5924.834,E2 -5924.834} C_VEL
LIN {X 0,Y 503.663,Z 541.434,A -85,B 0,C 180,E1 -5925.118,E2 -5925.118} C_VEL
LIN {X 0,Y 505.6,Z 553.985,A -85,B 0,C 180,E1 -5925.391,E2 -5925.391} C_VEL
LIN {X 0,Y 504.736,Z 652.384,A -85,B 0,C 180,E1 -5926.948,E2 -5926.948} C_VEL
LIN {X 0,Y 504.531,Z 666.167,A -85,B 0,C 180,E1 -5927.341,E2 -5927.341} C_VEL
LIN {X 0,Y 504.274,Z 678.457,A -85,B 0,C 180,E1 -5927.855,E2 -5927.855} C_VEL
LIN {X 0,Y 503.988,Z 690.605,A -85,B 0,C 180,E1 -5928.538,E2 -5928.538} C_VEL
LIN {X 0,Y 503.541,Z 701.86,A -85,B 0,C 180,E1 -5929.343,E2 -5929.343} C_VEL
LIN {X 0,Y 503.204,Z 712,A -85,B 0,C 180,E1 -5930.25,E2 -5930.25} C_VEL
LIN {X 0,Y 502.974,Z 720.32,A -85,B 0,C 180,E1 -5931.158,E2 -5931.158} C_VEL
LIN {X 0,Y 502.639,Z 729.37,A -85,B 0,C 180,E1 -5932.367,E2 -5932.367} C_VEL
LIN {X 0,Y 502.511,Z 736.632,A -85,B 0,C 180,E1 -5933.576,E2 -5933.576} C_VEL
LIN {X 0,Y 502.232,Z 742.448,A -85,B 0,C 180,E1 -5934.781,E2 -5934.781} C_VEL
LIN {X 0,Y 502.265,Z 747.021,A -85,B 0,C 180,E1 -5935.988,E2 -5935.988} C_VEL
LIN {X 0,Y 502.166,Z 749.441,A -85,B 0,C 180,E1 -5936.791,E2 -5936.791} C_VEL
LIN {X 0,Y 502.141,Z 751.41,A -85,B 0,C 180,E1 -5937.594,E2 -5937.594} C_VEL
LIN {X 0,Y 502.042,Z 752.959,A -85,B 0,C 180,E1 -5938.396,E2 -5938.396} C_VEL
LIN {X 0,Y 501.992,Z 754.088,A -85,B 0,C 180,E1 -5939.198,E2 -5939.198} C_VEL
LIN {X 0,Y 501.981,Z 754.792,A -85,B 0,C 180,E1 -5940,E2 -5940} C_VEL
LIN {X 0,Y 502.036,Z 755.015,A -85,B 0,C 180,E1 -5941.604,E2 -5941.604} C_VEL
LIN {X 0,Y 502.118,Z 754.534,A -85,B 0,C 180,E1 -5942.407,E2 -5942.407} C_VEL
LIN {X 0,Y 502.114,Z 753.644,A -85,B 0,C 180,E1 -5943.209,E2 -5943.209} C_VEL
LIN {X 0,Y 502.167,Z 752.331,A -85,B 0,C 180,E1 -5944.013,E2 -5944.013} C_VEL
LIN {X 0,Y 502.164,Z 749.6,A -85,B 0,C 180,E1 -5945.219,E2 -5945.219} C_VEL
LIN {X 0,Y 502.227,Z 744.49,A -85,B 0,C 180,E1 -5946.791,E2 -5946.791} C_VEL
LIN {X 0,Y 502.405,Z 737.982,A -85,B 0,C 180,E1 -5948.244,E2 -5948.244} C_VEL
LIN {X 0,Y 502.607,Z 731.041,A -85,B 0,C 180,E1 -5949.457,E2 -5949.457} C_VEL
LIN {X 0,Y 502.887,Z 722.38,A -85,B 0,C 180,E1 -5950.671,E2 -5950.671} C_VEL
LIN {X 0,Y 503.183,Z 712.315,A -85,B 0,C 180,E1 -5951.804,E2 -5951.804} C_VEL
LIN {X 0,Y 503.531,Z 702.717,A -85,B 0,C 180,E1 -5952.679,E2 -5952.679} C_VEL
LIN {X 0,Y 503.901,Z 691.353,A -85,B 0,C 180,E1 -5953.51,E2 -5953.51} C_VEL
LIN {X 0,Y 504.229,Z 678.899,A -85,B 0,C 180,E1 -5954.221,E2 -5954.221} C_VEL
LIN {X 0,Y 504.465,Z 667.069,A -85,B 0,C 180,E1 -5954.729,E2 -5954.729} C_VEL
LIN {X 0,Y 504.754,Z 654.314,A -85,B 0,C 180,E1 -5955.108,E2 -5955.108} C_VEL
LIN {X 0,Y 504.954,Z 635.147,A -85,B 0,C 180,E1 -5955.437,E2 -5955.437} C_VEL
LIN {X 0,Y 505.428,Z 553.249,A -85,B 0,C 180,E1 -5956.674,E2 -5956.674} C_VEL
LIN {X 0,Y 503.594,Z 541.296,A -85,B 0,C 180,E1 -5956.944,E2 -5956.944} C_VEL
LIN {X 0,Y 504.119,Z 524.084,A -85,B 0,C 180,E1 -5959.547,E2 -5959.547} C_VEL
LIN {X 0,Y 504.736,Z 504.727,A -85,B 0,C 180,E1 -5962.514,E2 -5962.514} C_VEL
LIN {X 0,Y 505.444,Z 486.568,A -85,B 0,C 180,E1 -5965.337,E2 -5965.337} C_VEL
LIN {X 0,Y 504.633,Z 481.155,A -85,B 0,C 180,E1 -5966.243,E2 -5966.243} C_VEL
LIN {X 0,Y 502.867,Z 472.975,A -85,B 0,C 180,E1 -5967.691,E2 -5967.691} C_VEL
LIN {X 0,Y 502.813,Z 472.977,A -85,B 0,C 180,E1 -5970.211,E2 -5970.211} C_VEL
LIN {X 0,Y 502.835,Z 472.974,A -85,B 0,C 180,E1 -5973.031,E2 -5973.031} C_VEL
LIN {X 0,Y 502.779,Z 472.981,A -85,B 0,C 180,E1 -5975.951,E2 -5975.951} C_VEL
LIN {X 0,Y 502.792,Z 472.976,A -85,B 0,C 180,E1 -5978.263,E2 -5978.263} C_VEL
LIN {X 0,Y 502.144,Z 473.057,A -85,B 0,C 180,E1 -5978.932,E2 -5978.932} C_VEL
LIN {X 0,Y 499.32,Z 473.415,A -85,B 0,C 180,E1 -5980.018,E2 -5980.018} C_VEL
LIN {X 0,Y 496.91,Z 473.72,A -85,B 0,C 180,E1 -5980.893,E2 -5980.893} C_VEL
LIN {X 0,Y 495.854,Z 473.848,A -85,B 0,C 180,E1 -5981.569,E2 -5981.569} C_VEL
LIN {X 0,Y 495.757,Z 473.857,A -85,B 0,C 180,E1 -5981.798,E2 -5981.798} C_VEL
LIN {X 0,Y 495.74,Z 473.856,A -85,B 0,C 180,E1 -5985.141,E2 -5985.141} C_VEL
LIN {X 0,Y 495.759,Z 473.852,A -85,B 0,C 180,E1 -5988.219,E2 -5988.219} C_VEL
LIN {X 0,Y 495.753,Z 473.858,A -85,B 0,C 180,E1 -5991.408,E2 -5991.408} C_VEL
LIN {X 0,Y 495.75,Z 473.852,A -85,B 0,C 180,E1 -5994.462,E2 -5994.462} C_VEL
LIN {X 0,Y 495.769,Z 473.856,A -85,B 0,C 180,E1 -5997.406,E2 -5997.406} C_VEL
LIN {X 0,Y 495.768,Z 473.85,A -85,B 0,C 180,E1 -6000.254,E2 -6000.254} C_VEL
LIN {X 0,Y 495.825,Z 473.847,A -85,B 0,C 180,E1 -6003.251,E2 -6003.251} C_VEL
LIN {X 0,Y 495.75,Z 473.858,A -85,B 0,C 180,E1 -6005.725,E2 -6005.725} C_VEL
LIN {X 0,Y 495.745,Z 473.853,A -85,B 0,C 180,E1 -6008.371,E2 -6008.371} C_VEL
LIN {X 0,Y 495.787,Z 473.849,A -85,B 0,C 180,E1 -6010.972,E2 -6010.972} C_VEL
LIN {X 0,Y 495.782,Z 473.857,A -85,B 0,C 180,E1 -6013.53,E2 -6013.53} C_VEL
LIN {X 0,Y 495.801,Z 473.847,A -85,B 0,C 180,E1 -6016.056,E2 -6016.056} C_VEL
LIN {X 0,Y 495.854,Z 473.839,A -85,B 0,C 180,E1 -6018.555,E2 -6018.555} C_VEL
LIN {X 0,Y 495.876,Z 473.84,A -85,B 0,C 180,E1 -6021.852,E2 -6021.852} C_VEL
LIN {X 0,Y 495.898,Z 473.834,A -85,B 0,C 180,E1 -6024.306,E2 -6024.306} C_VEL
LIN {X 0,Y 495.997,Z 473.829,A -85,B 0,C 180,E1 -6027.564,E2 -6027.564} C_VEL
LIN {X 0,Y 496.001,Z 473.823,A -85,B 0,C 180,E1 -6030,E2 -6030} C_VEL
LIN {X 0,Y 495.996,Z 473.821,A -85,B 0,C 180,E1 -6032.436,E2 -6032.436} C_VEL
LIN {X 0,Y 495.892,Z 473.839,A -85,B 0,C 180,E1 -6035.693,E2 -6035.693} C_VEL
LIN {X 0,Y 495.875,Z 473.837,A -85,B 0,C 180,E1 -6038.148,E2 -6038.148} C_VEL
LIN {X 0,Y 495.854,Z 473.848,A -85,B 0,C 180,E1 -6041.445,E2 -6041.445} C_VEL
LIN {X 0,Y 495.792,Z 473.848,A -85,B 0,C 180,E1 -6044.783,E2 -6044.783} C_VEL
LIN {X 0,Y 495.789,Z 473.855,A -85,B 0,C 180,E1 -6047.319,E2 -6047.319} C_VEL
LIN {X 0,Y 495.78,Z 473.851,A -85,B 0,C 180,E1 -6049.89,E2 -6049.89} C_VEL
LIN {X 0,Y 495.768,Z 473.852,A -85,B 0,C 180,E1 -6052.862,E2 -6052.862} C_VEL
LIN {X 0,Y 495.793,Z 473.848,A -85,B 0,C 180,E1 -6056.068,E2 -6056.068} C_VEL
LIN {X 0,Y 495.774,Z 473.851,A -85,B 0,C 180,E1 -6058.815,E2 -6058.815} C_VEL
LIN {X 0,Y 495.757,Z 473.855,A -85,B 0,C 180,E1 -6061.725,E2 -6061.725} C_VEL
LIN {X 0,Y 495.77,Z 473.851,A -85,B 0,C 180,E1 -6064.694,E2 -6064.694} C_VEL
LIN {X 0,Y 495.731,Z 473.86,A -85,B 0,C 180,E1 -6067.562,E2 -6067.562} C_VEL
LIN {X 0,Y 495.769,Z 473.851,A -85,B 0,C 180,E1 -6070.7,E2 -6070.7} C_VEL
LIN {X 0,Y 495.737,Z 473.857,A -85,B 0,C 180,E1 -6073.696,E2 -6073.696} C_VEL
LIN {X 0,Y 495.73,Z 473.854,A -85,B 0,C 180,E1 -6076.306,E2 -6076.306} C_VEL
LIN {X 0,Y 495.768,Z 473.859,A -85,B 0,C 180,E1 -6079.3,E2 -6079.3} C_VEL
LIN {X 0,Y 495.731,Z 473.855,A -85,B 0,C 180,E1 -6082.439,E2 -6082.439} C_VEL
LIN {X 0,Y 495.783,Z 473.856,A -85,B 0,C 180,E1 -6085.457,E2 -6085.457} C_VEL
LIN {X 0,Y 495.758,Z 473.852,A -85,B 0,C 180,E1 -6088.364,E2 -6088.364} C_VEL
LIN {X 0,Y 495.79,Z 473.852,A -85,B 0,C 180,E1 -6091.507,E2 -6091.507} C_VEL
LIN {X 0,Y 495.864,Z 474.018,A -85,B 0,C 180,E1 -6093.433,E2 -6093.433} C_VEL
LIN {X 0,Y 498.339,Z 486.583,A -85,B 0,C 180,E1 -6095.416,E2 -6095.416} C_VEL
LIN {X 0,Y 497.697,Z 509.324,A -85,B 0,C 180,E1 -6098.748,E2 -6098.748} C_VEL
LIN {X 0,Y 497.095,Z 530.741,A -85,B 0,C 180,E1 -6101.878,E2 -6101.878} C_VEL
LIN {X 0,Y 496.728,Z 545.531,A -85,B 0,C 180,E1 -6104.038,E2 -6104.038} C_VEL
LIN {X 0,Y 498.533,Z 557.62,A -85,B 0,C 180,E1 -6104.288,E2 -6104.288} C_VEL
LIN {X 0,Y 497.815,Z 655.451,A -85,B 0,C 180,E1 -6105.801,E2 -6105.801} C_VEL
LIN {X 0,Y 497.591,Z 668.353,A -85,B 0,C 180,E1 -6106.159,E2 -6106.159} C_VEL
LIN {X 0,Y 497.273,Z 680.735,A -85,B 0,C 180,E1 -6106.671,E2 -6106.671} C_VEL
LIN {X 0,Y 496.904,Z 693.41,A -85,B 0,C 180,E1 -6107.375,E2 -6107.375} C_VEL
LIN {X 0,Y 496.585,Z 704.242,A -85,B 0,C 180,E1 -6108.158,E2 -6108.158} C_VEL
LIN {X 0,Y 496.188,Z 715.559,A -85,B 0,C 180,E1 -6109.183,E2 -6109.183} C_VEL
LIN {X 0,Y 495.888,Z 724.663,A -85,B 0,C 180,E1 -6110.208,E2 -6110.208} C_VEL
LIN {X 0,Y 495.566,Z 733.475,A -85,B 0,C 180,E1 -6111.436,E2 -6111.436} C_VEL
LIN {X 0,Y 495.349,Z 740.57,A -85,B 0,C 180,E1 -6112.664,E2 -6112.664} C_VEL
LIN {X 0,Y 495.256,Z 746.216,A -85,B 0,C 180,E1 -6113.89,E2 -6113.89} C_VEL
LIN {X 0,Y 495.044,Z 750.637,A -85,B 0,C 180,E1 -6115.114,E2 -6115.114} C_VEL
LIN {X 0,Y 495.134,Z 752.955,A -85,B 0,C 180,E1 -6115.93,E2 -6115.93} C_VEL
LIN {X 0,Y 495.05,Z 754.854,A -85,B 0,C 180,E1 -6116.745,E2 -6116.745} C_VEL
LIN {X 0,Y 495.024,Z 756.318,A -85,B 0,C 180,E1 -6117.559,E2 -6117.559} C_VEL
LIN {X 0,Y 494.911,Z 757.973,A -85,B 0,C 180,E1 -6119.186,E2 -6119.186} C_VEL
LIN {X 0,Y 494.898,Z 758.223,A -85,B 0,C 180,E1 -6120,E2 -6120} C_VEL
LIN {X 0,Y 494.911,Z 758.037,A -85,B 0,C 180,E1 -6120.814,E2 -6120.814} C_VEL
LIN {X 0,Y 495.024,Z 756.471,A -85,B 0,C 180,E1 -6122.441,E2 -6122.441} C_VEL
LIN {X 0,Y 495.05,Z 755.085,A -85,B 0,C 180,E1 -6123.255,E2 -6123.255} C_VEL
LIN {X 0,Y 495.082,Z 752.175,A -85,B 0,C 180,E1 -6124.478,E2 -6124.478} C_VEL
LIN {X 0,Y 495.223,Z 748.209,A -85,B 0,C 180,E1 -6125.701,E2 -6125.701} C_VEL
LIN {X 0,Y 495.318,Z 742.173,A -85,B 0,C 180,E1 -6127.111,E2 -6127.111} C_VEL
LIN {X 0,Y 495.524,Z 735.37,A -85,B 0,C 180,E1 -6128.359,E2 -6128.359} C_VEL
LIN {X 0,Y 495.762,Z 726.968,A -85,B 0,C 180,E1 -6129.588,E2 -6129.588} C_VEL
LIN {X 0,Y 496.046,Z 718.328,A -85,B 0,C 180,E1 -6130.614,E2 -6130.614} C_VEL
LIN {X 0,Y 496.453,Z 707.697,A -85,B 0,C 180,E1 -6131.638,E2 -6131.638} C_VEL
LIN {X 0,Y 496.808,Z 696.566,A -85,B 0,C 180,E1 -6132.488,E2 -6132.488} C_VEL
LIN {X 0,Y 497.093,Z 685.143,A -85,B 0,C 180,E1 -6133.178,E2 -6133.178} C_VEL
LIN {X 0,Y 497.404,Z 672.818,A -85,B 0,C 180,E1 -6133.742,E2 -6133.742} C_VEL
LIN {X 0,Y 497.709,Z 659.042,A -85,B 0,C 180,E1 -6134.176,E2 -6134.176} C_VEL
LIN {X 0,Y 497.854,Z 645.344,A -85,B 0,C 180,E1 -6134.433,E2 -6134.433} C_VEL
LIN {X 0,Y 498.468,Z 556.739,A -85,B 0,C 180,E1 -6135.807,E2 -6135.807} C_VEL
LIN {X 0,Y 496.748,Z 545.815,A -85,B 0,C 180,E1 -6136.064,E2 -6136.064} C_VEL
LIN {X 0,Y 497.237,Z 523.929,A -85,B 0,C 180,E1 -6139.185,E2 -6139.185} C_VEL
LIN {X 0,Y 497.65,Z 504.154,A -85,B 0,C 180,E1 -6141.978,E2 -6141.978} C_VEL
LIN {X 0,Y 498.029,Z 486.863,A -85,B 0,C 180,E1 -6144.379,E2 -6144.379} C_VEL
LIN {X 0,Y 497.199,Z 480.347,A -85,B 0,C 180,E1 -6145.321,E2 -6145.321} C_VEL
LIN {X 0,Y 495.831,Z 473.851,A -85,B 0,C 180,E1 -6146.295,E2 -6146.295} C_VEL
LIN {X 0,Y 495.775,Z 473.858,A -85,B 0,C 180,E1 -6148.815,E2 -6148.815} C_VEL
LIN {X 0,Y 495.758,Z 473.857,A -85,B 0,C 180,E1 -6151.725,E2 -6151.725} C_VEL
LIN {X 0,Y 495.772,Z 473.858,A -85,B 0,C 180,E1 -6154.694,E2 -6154.694} C_VEL
LIN {X 0,Y 495.732,Z 473.857,A -85,B 0,C 180,E1 -6157.562,E2 -6157.562} C_VEL
LIN {X 0,Y 495.768,Z 473.857,A -85,B 0,C 180,E1 -6160.7,E2 -6160.7} C_VEL
LIN {X 0,Y 495.736,Z 473.857,A -85,B 0,C 180,E1 -6164.001,E2 -6164.001} C_VEL
LIN {X 0,Y 495.736,Z 473.857,A -85,B 0,C 180,E1 -6167.118,E2 -6167.118} C_VEL
LIN {X 0,Y 495.761,Z 473.855,A -85,B 0,C 180,E1 -6169.953,E2 -6169.953} C_VEL
LIN {X 0,Y 495.733,Z 473.86,A -85,B 0,C 180,E1 -6172.553,E2 -6172.553} C_VEL
LIN {X 0,Y 495.786,Z 473.85,A -85,B 0,C 180,E1 -6175.457,E2 -6175.457} C_VEL
LIN {X 0,Y 495.763,Z 473.859,A -85,B 0,C 180,E1 -6178.364,E2 -6178.364} C_VEL
LIN {X 0,Y 495.792,Z 473.851,A -85,B 0,C 180,E1 -6181.506,E2 -6181.506} C_VEL
LIN {X 0,Y 495.843,Z 473.973,A -85,B 0,C 180,E1 -6183.603,E2 -6183.603} C_VEL
LIN {X 0,Y 498.938,Z 487.34,A -85,B 0,C 180,E1 -6185.669,E2 -6185.669} C_VEL
LIN {X 0,Y 499.131,Z 490.776,A -85,B 0,C 180,E1 -6186.154,E2 -6186.154} C_VEL
LIN {X 0,Y 498.033,Z 515.922,A -85,B 0,C 180,E1 -6189.558,E2 -6189.558} C_VEL
LIN {X 0,Y 497.711,Z 524.389,A -85,B 0,C 180,E1 -6190.692,E2 -6190.692} C_VEL
LIN {X 0,Y 499.942,Z 539.15,A -85,B 0,C 180,E1 -6191.029,E2 -6191.029} C_VEL
LIN {X 0,Y 498.882,Z 661.397,A -85,B 0,C 180,E1 -6192.879,E2 -6192.879} C_VEL
LIN {X 0,Y 498.575,Z 675.729,A -85,B 0,C 180,E1 -6193.246,E2 -6193.246} C_VEL
LIN {X 0,Y 498.296,Z 689.367,A -85,B 0,C 180,E1 -6193.762,E2 -6193.762} C_VEL
LIN {X 0,Y 497.866,Z 701.078,A -85,B 0,C 180,E1 -6194.338,E2 -6194.338} C_VEL
LIN {X 0,Y 497.331,Z 714.184,A -85,B 0,C 180,E1 -6195.159,E2 -6195.159} C_VEL
LIN {X 0,Y 496.862,Z 726.066,A -85,B 0,C 180,E1 -6196.086,E2 -6196.086} C_VEL
LIN {X 0,Y 496.433,Z 736.919,A -85,B 0,C 180,E1 -6197.116,E2 -6197.116} C_VEL
LIN {X 0,Y 496.11,Z 746.342,A -85,B 0,C 180,E1 -6198.189,E2 -6198.189} C_VEL
LIN {X 0,Y 495.746,Z 755.116,A -85,B 0,C 180,E1 -6199.38,E2 -6199.38} C_VEL
LIN {X 0,Y 495.446,Z 763.82,A -85,B 0,C 180,E1 -6200.817,E2 -6200.817} C_VEL
LIN {X 0,Y 495.214,Z 770.827,A -85,B 0,C 180,E1 -6202.252,E2 -6202.252} C_VEL
LIN {X 0,Y 495.117,Z 776.666,A -85,B 0,C 180,E1 -6203.764,E2 -6203.764} C_VEL
LIN {X 0,Y 495.031,Z 780.646,A -85,B 0,C 180,E1 -6205.114,E2 -6205.114} C_VEL
LIN {X 0,Y 495.033,Z 784.114,A -85,B 0,C 180,E1 -6206.745,E2 -6206.745} C_VEL
LIN {X 0,Y 494.959,Z 786.16,A -85,B 0,C 180,E1 -6208.373,E2 -6208.373} C_VEL
LIN {X 0,Y 494.896,Z 786.834,A -85,B 0,C 180,E1 -6210,E2 -6210} C_VEL
LIN {X 0,Y 494.959,Z 786.145,A -85,B 0,C 180,E1 -6211.627,E2 -6211.627} C_VEL
LIN {X 0,Y 495.033,Z 784.083,A -85,B 0,C 180,E1 -6213.256,E2 -6213.256} C_VEL
LIN {X 0,Y 495.031,Z 780.594,A -85,B 0,C 180,E1 -6214.887,E2 -6214.887} C_VEL
LIN {X 0,Y 495.117,Z 776.579,A -85,B 0,C 180,E1 -6216.235,E2 -6216.235} C_VEL
LIN {X 0,Y 495.214,Z 770.702,A -85,B 0,C 180,E1 -6217.748,E2 -6217.748} C_VEL
LIN {X 0,Y 495.446,Z 763.649,A -85,B 0,C 180,E1 -6219.183,E2 -6219.183} C_VEL
LIN {X 0,Y 495.736,Z 754.868,A -85,B 0,C 180,E1 -6220.62,E2 -6220.62} C_VEL
LIN {X 0,Y 496.099,Z 745.164,A -85,B 0,C 180,E1 -6221.916,E2 -6221.916} C_VEL
LIN {X 0,Y 496.51,Z 734.475,A -85,B 0,C 180,E1 -6223.09,E2 -6223.09} C_VEL
LIN {X 0,Y 496.932,Z 723.023,A -85,B 0,C 180,E1 -6224.121,E2 -6224.121} C_VEL
LIN {X 0,Y 497.382,Z 711.911,A -85,B 0,C 180,E1 -6224.944,E2 -6224.944} C_VEL
LIN {X 0,Y 497.866,Z 698.195,A -85,B 0,C 180,E1 -6225.755,E2 -6225.755} C_VEL
LIN {X 0,Y 498.232,Z 684.285,A -85,B 0,C 180,E1 -6226.387,E2 -6226.387} C_VEL
LIN {X 0,Y 498.562,Z 670.441,A -85,B 0,C 180,E1 -6226.842,E2 -6226.842} C_VEL
LIN {X 0,Y 498.837,Z 655.733,A -85,B 0,C 180,E1 -6227.151,E2 -6227.151} C_VEL
LIN {X 0,Y 499.798,Z 538.871,A -85,B 0,C 180,E1 -6228.923,E2 -6228.923} C_VEL
LIN {X 0,Y 497.705,Z 524.843,A -85,B 0,C 180,E1 -6229.238,E2 -6229.238} C_VEL
LIN {X 0,Y 498.848,Z 498.769,A -85,B 0,C 180,E1 -6232.795,E2 -6232.795} C_VEL
LIN {X 0,Y 499.361,Z 489.555,A -85,B 0,C 180,E1 -6234.089,E2 -6234.089} C_VEL
LIN {X 0,Y 496.79,Z 477.656,A -85,B 0,C 180,E1 -6236.012,E2 -6236.012} C_VEL
LIN {X 0,Y 495.833,Z 473.849,A -85,B 0,C 180,E1 -6236.664,E2 -6236.664} C_VEL
LIN {X 0,Y 495.769,Z 473.86,A -85,B 0,C 180,E1 -6239.746,E2 -6239.746} C_VEL
LIN {X 0,Y 495.771,Z 473.854,A -85,B 0,C 180,E1 -6242.594,E2 -6242.594} C_VEL
LIN {X 0,Y 495.75,Z 473.86,A -85,B 0,C 180,E1 -6245.538,E2 -6245.538} C_VEL
LIN {X 0,Y 495.766,Z 473.856,A -85,B 0,C 180,E1 -6248.768,E2 -6248.768} C_VEL
LIN {X 0,Y 495.78,Z 473.852,A -85,B 0,C 180,E1 -6251.779,E2 -6251.779} C_VEL
LIN {X 0,Y 495.752,Z 473.86,A -85,B 0,C 180,E1 -6255.14,E2 -6255.14} C_VEL
LIN {X 0,Y 495.759,Z 473.854,A -85,B 0,C 180,E1 -6258.219,E2 -6258.219} C_VEL
LIN {X 0,Y 495.754,Z 473.858,A -85,B 0,C 180,E1 -6261.409,E2 -6261.409} C_VEL
LIN {X 0,Y 495.753,Z 473.859,A -85,B 0,C 180,E1 -6264.463,E2 -6264.463} C_VEL
LIN {X 0,Y 495.772,Z 473.855,A -85,B 0,C 180,E1 -6267.406,E2 -6267.406} C_VEL
LIN {X 0,Y 495.77,Z 473.858,A -85,B 0,C 180,E1 -6270.254,E2 -6270.254} C_VEL
LIN {X 0,Y 495.827,Z 473.855,A -85,B 0,C 180,E1 -6273.251,E2 -6273.251} C_VEL
LIN {X 0,Y 495.853,Z 473.93,A -85,B 0,C 180,E1 -6273.992,E2 -6273.992} C_VEL
LIN {X 0,Y 498.662,Z 486.906,A -85,B 0,C 180,E1 -6276.362,E2 -6276.362} C_VEL
LIN {X 0,Y 498.367,Z 496.043,A -85,B 0,C 180,E1 -6277.838,E2 -6277.838} C_VEL
LIN {X 0,Y 497.462,Z 517.249,A -85,B 0,C 180,E1 -6281.185,E2 -6281.185} C_VEL
LIN {X 0,Y 496.74,Z 539.478,A -85,B 0,C 180,E1 -6284.616,E2 -6284.616} C_VEL
LIN {X 0,Y 496.713,Z 541.138,A -85,B 0,C 180,E1 -6284.852,E2 -6284.852} C_VEL
LIN {X 0,Y 498.755,Z 554.05,A -85,B 0,C 180,E1 -6285.15,E2 -6285.15} C_VEL
LIN {X 0,Y 498.024,Z 639.617,A -85,B 0,C 180,E1 -6286.535,E2 -6286.535} C_VEL
LIN {X 0,Y 497.799,Z 655.896,A -85,B 0,C 180,E1 -6286.841,E2 -6286.841} C_VEL
LIN {X 0,Y 497.579,Z 668.481,A -85,B 0,C 180,E1 -6287.243,E2 -6287.243} C_VEL
LIN {X 0,Y 497.228,Z 682.083,A -85,B 0,C 180,E1 -6287.863,E2 -6287.863} C_VEL
LIN {X 0,Y 496.928,Z 693.839,A -85,B 0,C 180,E1 -6288.58,E2 -6288.58} C_VEL
LIN {X 0,Y 496.429,Z 705.613,A -85,B 0,C 180,E1 -6289.498,E2 -6289.498} C_VEL
LIN {X 0,Y 496.161,Z 715.112,A -85,B 0,C 180,E1 -6290.419,E2 -6290.419} C_VEL
LIN {X 0,Y 495.817,Z 723.783,A -85,B 0,C 180,E1 -6291.441,E2 -6291.441} C_VEL
LIN {X 0,Y 495.52,Z 732.182,A -85,B 0,C 180,E1 -6292.666,E2 -6292.666} C_VEL
LIN {X 0,Y 495.433,Z 738.934,A -85,B 0,C 180,E1 -6293.893,E2 -6293.893} C_VEL
LIN {X 0,Y 495.114,Z 744.326,A -85,B 0,C 180,E1 -6295.114,E2 -6295.114} C_VEL
LIN {X 0,Y 495.127,Z 748.522,A -85,B 0,C 180,E1 -6296.338,E2 -6296.338} C_VEL
LIN {X 0,Y 495.074,Z 751.652,A -85,B 0,C 180,E1 -6297.559,E2 -6297.559} C_VEL
LIN {X 0,Y 494.969,Z 753.207,A -85,B 0,C 180,E1 -6298.373,E2 -6298.373} C_VEL
LIN {X 0,Y 494.912,Z 754.327,A -85,B 0,C 180,E1 -6299.186,E2 -6299.186} C_VEL
LIN {X 0,Y 494.91,Z 755.327,A -85,B 0,C 180,E1 -6300.814,E2 -6300.814} C_VEL
LIN {X 0,Y 494.963,Z 755.242,A -85,B 0,C 180,E1 -6301.627,E2 -6301.627} C_VEL
LIN {X 0,Y 495.022,Z 754.75,A -85,B 0,C 180,E1 -6302.441,E2 -6302.441} C_VEL
LIN {X 0,Y 495.038,Z 753.832,A -85,B 0,C 180,E1 -6303.255,E2 -6303.255} C_VEL
LIN {X 0,Y 495.065,Z 752.513,A -85,B 0,C 180,E1 -6304.07,E2 -6304.07} C_VEL
LIN {X 0,Y 495.102,Z 749.743,A -85,B 0,C 180,E1 -6305.294,E2 -6305.294} C_VEL
LIN {X 0,Y 495.144,Z 745.087,A -85,B 0,C 180,E1 -6306.749,E2 -6306.749} C_VEL
LIN {X 0,Y 495.26,Z 740.982,A -85,B 0,C 180,E1 -6307.748,E2 -6307.748} C_VEL
LIN {X 0,Y 495.461,Z 734.737,A -85,B 0,C 180,E1 -6308.977,E2 -6308.977} C_VEL
LIN {X 0,Y 495.679,Z 726.947,A -85,B 0,C 180,E1 -6310.209,E2 -6310.209} C_VEL
LIN {X 0,Y 496.101,Z 717.156,A -85,B 0,C 180,E1 -6311.439,E2 -6311.439} C_VEL
LIN {X 0,Y 496.326,Z 708.126,A -85,B 0,C 180,E1 -6312.367,E2 -6312.367} C_VEL
LIN {X 0,Y 496.763,Z 696.985,A -85,B 0,C 180,E1 -6313.291,E2 -6313.291} C_VEL
LIN {X 0,Y 497.171,Z 684.302,A -85,B 0,C 180,E1 -6314.114,E2 -6314.114} C_VEL
LIN {X 0,Y 497.504,Z 671.73,A -85,B 0,C 180,E1 -6314.731,E2 -6314.731} C_VEL
LIN {X 0,Y 497.716,Z 659.275,A -85,B 0,C 180,E1 -6315.169,E2 -6315.169} C_VEL
LIN {X 0,Y 497.951,Z 645.509,A -85,B 0,C 180,E1 -6315.476,E2 -6315.476} C_VEL
LIN {X 0,Y 498.632,Z 554.023,A -85,B 0,C 180,E1 -6316.897,E2 -6316.897} C_VEL
LIN {X 0,Y 496.612,Z 541.273,A -85,B 0,C 180,E1 -6317.18,E2 -6317.18} C_VEL
LIN {X 0,Y 497.186,Z 523.979,A -85,B 0,C 180,E1 -6319.831,E2 -6319.831} C_VEL
LIN {X 0,Y 497.836,Z 505.989,A -85,B 0,C 180,E1 -6322.625,E2 -6322.625} C_VEL
LIN {X 0,Y 498.586,Z 488.276,A -85,B 0,C 180,E1 -6325.416,E2 -6325.416} C_VEL
LIN {X 0,Y 497.693,Z 482.404,A -85,B 0,C 180,E1 -6326.412,E2 -6326.412} C_VEL
LIN {X 0,Y 495.831,Z 473.851,A -85,B 0,C 180,E1 -6327.936,E2 -6327.936} C_VEL
LIN {X 0,Y 495.755,Z 473.855,A -85,B 0,C 180,E1 -6330.687,E2 -6330.687} C_VEL
LIN {X 0,Y 495.764,Z 473.859,A -85,B 0,C 180,E1 -6333.564,E2 -6333.564} C_VEL
LIN {X 0,Y 495.732,Z 473.854,A -85,B 0,C 180,E1 -6336.544,E2 -6336.544} C_VEL
LIN {X 0,Y 495.759,Z 473.859,A -85,B 0,C 180,E1 -6339.638,E2 -6339.638} C_VEL
LIN {X 0,Y 495.757,Z 473.857,A -85,B 0,C 180,E1 -6341.798,E2 -6341.798} C_VEL
LIN {X 0,Y 495.064,Z 473.94,A -85,B 0,C 180,E1 -6342.476,E2 -6342.476} C_VEL
LIN {X 0,Y 492.215,Z 474.301,A -85,B 0,C 180,E1 -6343.577,E2 -6343.577} C_VEL
LIN {X 0,Y 489.817,Z 474.598,A -85,B 0,C 180,E1 -6344.465,E2 -6344.465} C_VEL
LIN {X 0,Y 488.782,Z 474.723,A -85,B 0,C 180,E1 -6345.15,E2 -6345.15} C_VEL
LIN {X 0,Y 488.694,Z 474.733,A -85,B 0,C 180,E1 -6345.382,E2 -6345.382} C_VEL
LIN {X 0,Y 488.71,Z 474.729,A -85,B 0,C 180,E1 -6348.584,E2 -6348.584} C_VEL
LIN {X 0,Y 488.706,Z 474.731,A -85,B 0,C 180,E1 -6350.947,E2 -6350.947} C_VEL
LIN {X 0,Y 488.679,Z 474.737,A -85,B 0,C 180,E1 -6353.868,E2 -6353.868} C_VEL
LIN {X 0,Y 488.74,Z 474.726,A -85,B 0,C 180,E1 -6356.877,E2 -6356.877} C_VEL
LIN {X 0,Y 488.726,Z 474.732,A -85,B 0,C 180,E1 -6359.781,E2 -6359.781} C_VEL
LIN {X 0,Y 488.794,Z 474.721,A -85,B 0,C 180,E1 -6363.056,E2 -6363.056} C_VEL
LIN {X 0,Y 488.691,Z 474.732,A -85,B 0,C 180,E1 -6366.254,E2 -6366.254} C_VEL
LIN {X 0,Y 488.748,Z 474.728,A -85,B 0,C 180,E1 -6369.176,E2 -6369.176} C_VEL
LIN {X 0,Y 488.761,Z 474.73,A -85,B 0,C 180,E1 -6371.628,E2 -6371.628} C_VEL
LIN {X 0,Y 488.767,Z 474.724,A -85,B 0,C 180,E1 -6375,E2 -6375} C_VEL
LIN {X 0,Y 488.808,Z 474.717,A -85,B 0,C 180,E1 -6378.387,E2 -6378.387} C_VEL
LIN {X 0,Y 488.821,Z 474.72,A -85,B 0,C 180,E1 -6381.734,E2 -6381.734} C_VEL
LIN {X 0,Y 488.857,Z 474.711,A -85,B 0,C 180,E1 -6384.224,E2 -6384.224} C_VEL
LIN {X 0,Y 488.964,Z 474.705,A -85,B 0,C 180,E1 -6387.529,E2 -6387.529} C_VEL
LIN {X 0,Y 488.957,Z 474.7,A -85,B 0,C 180,E1 -6390.824,E2 -6390.824} C_VEL
LIN {X 0,Y 488.964,Z 474.697,A -85,B 0,C 180,E1 -6392.471,E2 -6392.471} C_VEL
LIN {X 0,Y 488.85,Z 474.715,A -85,B 0,C 180,E1 -6395.776,E2 -6395.776} C_VEL
LIN {X 0,Y 488.819,Z 474.716,A -85,B 0,C 180,E1 -6398.266,E2 -6398.266} C_VEL
LIN {X 0,Y 488.807,Z 474.723,A -85,B 0,C 180,E1 -6401.612,E2 -6401.612} C_VEL
LIN {X 0,Y 488.764,Z 474.726,A -85,B 0,C 180,E1 -6405,E2 -6405} C_VEL
LIN {X 0,Y 488.757,Z 474.723,A -85,B 0,C 180,E1 -6408.442,E2 -6408.442} C_VEL
LIN {X 0,Y 488.709,Z 474.733,A -85,B 0,C 180,E1 -6411.071,E2 -6411.071} C_VEL
LIN {X 0,Y 488.696,Z 474.734,A -85,B 0,C 180,E1 -6413.745,E2 -6413.745} C_VEL
LIN {X 0,Y 488.794,Z 474.722,A -85,B 0,C 180,E1 -6416.944,E2 -6416.944} C_VEL
LIN {X 0,Y 488.711,Z 474.729,A -85,B 0,C 180,E1 -6420.363,E2 -6420.363} C_VEL
LIN {X 0,Y 488.736,Z 474.733,A -85,B 0,C 180,E1 -6423.484,E2 -6423.484} C_VEL
LIN {X 0,Y 488.684,Z 474.732,A -85,B 0,C 180,E1 -6426.355,E2 -6426.355} C_VEL
LIN {X 0,Y 488.703,Z 474.738,A -85,B 0,C 180,E1 -6429.254,E2 -6429.254} C_VEL
LIN {X 0,Y 488.726,Z 474.732,A -85,B 0,C 180,E1 -6431.602,E2 -6431.602} C_VEL
LIN {X 0,Y 488.714,Z 474.731,A -85,B 0,C 180,E1 -6434.801,E2 -6434.801} C_VEL
LIN {X 0,Y 488.693,Z 474.737,A -85,B 0,C 180,E1 -6437.475,E2 -6437.475} C_VEL
LIN {X 0,Y 488.735,Z 474.729,A -85,B 0,C 180,E1 -6439.677,E2 -6439.677} C_VEL
LIN {X 0,Y 488.681,Z 474.735,A -85,B 0,C 180,E1 -6442.841,E2 -6442.841} C_VEL
LIN {X 0,Y 488.734,Z 474.727,A -85,B 0,C 180,E1 -6445.887,E2 -6445.887} C_VEL
LIN {X 0,Y 488.694,Z 474.735,A -85,B 0,C 180,E1 -6448.82,E2 -6448.82} C_VEL
LIN {X 0,Y 488.747,Z 474.729,A -85,B 0,C 180,E1 -6451.671,E2 -6451.671} C_VEL
LIN {X 0,Y 488.79,Z 474.796,A -85,B 0,C 180,E1 -6453.205,E2 -6453.205} C_VEL
LIN {X 0,Y 491.42,Z 487.772,A -85,B 0,C 180,E1 -6455.272,E2 -6455.272} C_VEL
LIN {X 0,Y 490.881,Z 507.189,A -85,B 0,C 180,E1 -6458.146,E2 -6458.146} C_VEL
LIN {X 0,Y 490.234,Z 529.457,A -85,B 0,C 180,E1 -6461.427,E2 -6461.427} C_VEL
LIN {X 0,Y 489.78,Z 545.718,A -85,B 0,C 180,E1 -6463.808,E2 -6463.808} C_VEL
LIN {X 0,Y 491.662,Z 557.674,A -85,B 0,C 180,E1 -6464.062,E2 -6464.062} C_VEL
LIN {X 0,Y 490.928,Z 654.649,A -85,B 0,C 180,E1 -6465.597,E2 -6465.597} C_VEL
LIN {X 0,Y 490.675,Z 667.894,A -85,B 0,C 180,E1 -6465.96,E2 -6465.96} C_VEL
LIN {X 0,Y 490.325,Z 680.454,A -85,B 0,C 180,E1 -6466.478,E2 -6466.478} C_VEL
LIN {X 0,Y 489.983,Z 692.2,A -85,B 0,C 180,E1 -6467.13,E2 -6467.13} C_VEL
LIN {X 0,Y 489.729,Z 702.868,A -85,B 0,C 180,E1 -6467.885,E2 -6467.885} C_VEL
LIN {X 0,Y 489.28,Z 713.443,A -85,B 0,C 180,E1 -6468.819,E2 -6468.819} C_VEL
LIN {X 0,Y 488.963,Z 722.971,A -85,B 0,C 180,E1 -6469.859,E2 -6469.859} C_VEL
LIN {X 0,Y 488.617,Z 730.804,A -85,B 0,C 180,E1 -6470.897,E2 -6470.897} C_VEL
LIN {X 0,Y 488.363,Z 738.464,A -85,B 0,C 180,E1 -6472.142,E2 -6472.142} C_VEL
LIN {X 0,Y 488.183,Z 744.572,A -85,B 0,C 180,E1 -6473.387,E2 -6473.387} C_VEL
LIN {X 0,Y 488.074,Z 749.409,A -85,B 0,C 180,E1 -6474.629,E2 -6474.629} C_VEL
LIN {X 0,Y 488.034,Z 753.116,A -85,B 0,C 180,E1 -6475.871,E2 -6475.871} C_VEL
LIN {X 0,Y 487.978,Z 755.023,A -85,B 0,C 180,E1 -6476.697,E2 -6476.697} C_VEL
